LIN {X 0,Y 529.01,Z 397.613,A -85,B 0,C 180,E1 4371.131,E2 4371.131} C_VEL
LIN {X 0,Y 529.22,Z 392.744,A -85,B 0,C 180,E1 4373.977,E2 4373.977} C_VEL
LIN {X 0,Y 529.564,Z 381.839,A -85,B 0,C 180,E1 4376.861,E2 4376.861} C_VEL
LIN {X 0,Y 530.019,Z 365.768,A -85,B 0,C 180,E1 4379.389,E2 4379.389} C_VEL
LIN {X 0,Y 530.692,Z 344.7,A -85,B 0,C 180,E1 4381.518,E2 4381.518} C_VEL
LIN {X 0,Y 531.24,Z 320.224,A -85,B 0,C 180,E1 4383.087,E2 4383.087} C_VEL
LIN {X 0,Y 530.045,Z 304.294,A -85,B 0,C 180,E1 4383.791,E2 4383.791} C_VEL
LIN {X 0,Y 528.638,Z 297.81,A -85,B 0,C 180,E1 4384.104,E2 4384.104} C_VEL
LIN {X 0,Y 528.492,Z 297.81,A -85,B 0,C 180,E1 4390.468,E2 4390.468} C_VEL
LIN {X 0,Y 528.252,Z 297.81,A -85,B 0,C 180,E1 4395.103,E2 4395.103} C_VEL
LIN {X 0,Y 528.481,Z 297.81,A -85,B 0,C 180,E1 4400.136,E2 4400.136} C_VEL
LIN {X 0,Y 528.543,Z 297.81,A -85,B 0,C 180,E1 4402,E2 4402} C_VEL
LIN {X 0,Y 531.152,Z 316.99,A -85,B 0,C 180,E1 4402.758,E2 4402.758} C_VEL
LIN {X 0,Y 530.693,Z 340.931,A -85,B 0,C 180,E1 4404.146,E2 4404.146} C_VEL
LIN {X 0,Y 530.077,Z 362.098,A -85,B 0,C 180,E1 4406.102,E2 4406.102} C_VEL
LIN {X 0,Y 529.641,Z 379.29,A -85,B 0,C 180,E1 4408.572,E2 4408.572} C_VEL
LIN {X 0,Y 529.309,Z 390.67,A -85,B 0,C 180,E1 4411.226,E2 4411.226} C_VEL
LIN {X 0,Y 529.244,Z 396.059,A -85,B 0,C 180,E1 4413.495,E2 4413.495} C_VEL
LIN {X 0,Y 529.086,Z 397.913,A -85,B 0,C 180,E1 4416.551,E2 4416.551} C_VEL
LIN {X 0,Y 529.245,Z 394.993,A -85,B 0,C 180,E1 4419.023,E2 4419.023} C_VEL
LIN {X 0,Y 529.429,Z 386.158,A -85,B 0,C 180,E1 4421.926,E2 4421.926} C_VEL
LIN {X 0,Y 529.791,Z 372.114,A -85,B 0,C 180,E1 4424.519,E2 4424.519} C_VEL
LIN {X 0,Y 530.286,Z 353.941,A -85,B 0,C 180,E1 4426.675,E2 4426.675} C_VEL
LIN {X 0,Y 530.924,Z 331.466,A -85,B 0,C 180,E1 4428.405,E2 4428.405} C_VEL
LIN {X 0,Y 530.572,Z 307.156,A -85,B 0,C 180,E1 4429.557,E2 4429.557} C_VEL
LIN {X 0,Y 528.62,Z 297.81,A -85,B 0,C 180,E1 4429.894,E2 4429.894} C_VEL
LIN {X 0,Y 528.216,Z 297.81,A -85,B 0,C 180,E1 4435.374,E2 4435.374} C_VEL
LIN {X 0,Y 528.104,Z 297.81,A -85,B 0,C 180,E1 4440.972,E2 4440.972} C_VEL
LIN {X 0,Y 528.237,Z 297.81,A -85,B 0,C 180,E1 4446.863,E2 4446.863} C_VEL
LIN {X 0,Y 528.018,Z 297.81,A -85,B 0,C 180,E1 4451.992,E2 4451.992} C_VEL
LIN {X 0,Y 528.084,Z 297.81,A -85,B 0,C 180,E1 4457.984,E2 4457.984} C_VEL
LIN {X 0,Y 528.182,Z 297.81,A -85,B 0,C 180,E1 4463.126,E2 4463.126} C_VEL
LIN {X 0,Y 528.097,Z 297.81,A -85,B 0,C 180,E1 4469.034,E2 4469.034} C_VEL
LIN {X 0,Y 528.212,Z 297.81,A -85,B 0,C 180,E1 4474.614,E2 4474.614} C_VEL
LIN {X 0,Y 528.506,Z 297.81,A -85,B 0,C 180,E1 4480.429,E2 4480.429} C_VEL
LIN {X 0,Y 528.221,Z 297.81,A -85,B 0,C 180,E1 4486.241,E2 4486.241} C_VEL
LIN {X 0,Y 528.457,Z 297.81,A -85,B 0,C 180,E1 4491.781,E2 4491.781} C_VEL
LIN {X 0,Y 528.654,Z 297.81,A -85,B 0,C 180,E1 4497.505,E2 4497.505} C_VEL
LIN {X 0,Y 528.738,Z 297.81,A -85,B 0,C 180,E1 4503.262,E2 4503.262} C_VEL
LIN {X 0,Y 528.535,Z 297.81,A -85,B 0,C 180,E1 4509.854,E2 4509.854} C_VEL
LIN {X 0,Y 528.47,Z 297.81,A -85,B 0,C 180,E1 4514.881,E2 4514.881} C_VEL
LIN {X 0,Y 528.387,Z 297.81,A -85,B 0,C 180,E1 4520.031,E2 4520.031} C_VEL
LIN {X 0,Y 528.213,Z 297.81,A -85,B 0,C 180,E1 4525.363,E2 4525.363} C_VEL
LIN {X 0,Y 528.113,Z 297.81,A -85,B 0,C 180,E1 4530.531,E2 4530.531} C_VEL
LIN {X 0,Y 525.63,Z 297.81,A -85,B 0,C 180,E1 4531.933,E2 4531.933} C_VEL
LIN {X 0,Y 520.125,Z 297.81,A -85,B 0,C 180,E1 4534.278,E2 4534.278} C_VEL
LIN {X 0,Y 520.117,Z 297.81,A -85,B 0,C 180,E1 4539.652,E2 4539.652} C_VEL
LIN {X 0,Y 520.204,Z 297.81,A -85,B 0,C 180,E1 4545.878,E2 4545.878} C_VEL
LIN {X 0,Y 520.222,Z 297.81,A -85,B 0,C 180,E1 4551.539,E2 4551.539} C_VEL
LIN {X 0,Y 520.219,Z 297.81,A -85,B 0,C 180,E1 4557.251,E2 4557.251} C_VEL
LIN {X 0,Y 520.326,Z 297.81,A -85,B 0,C 180,E1 4562.353,E2 4562.353} C_VEL
LIN {X 0,Y 520.675,Z 298.125,A -85,B 0,C 180,E1 4565.62,E2 4565.62} C_VEL
LIN {X 0,Y 526.8,Z 321.24,A -85,B 0,C 180,E1 4566.185,E2 4566.185} C_VEL
LIN {X 0,Y 526.441,Z 376.223,A -85,B 0,C 180,E1 4567.058,E2 4567.058} C_VEL
LIN {X 0,Y 525.477,Z 410.152,A -85,B 0,C 180,E1 4568.241,E2 4568.241} C_VEL
LIN {X 0,Y 524.336,Z 441.478,A -85,B 0,C 180,E1 4570.016,E2 4570.016} C_VEL
LIN {X 0,Y 523.111,Z 470.478,A -85,B 0,C 180,E1 4572.38,E2 4572.38} C_VEL
LIN {X 0,Y 522.191,Z 495.428,A -85,B 0,C 180,E1 4575.203,E2 4575.203} C_VEL
LIN {X 0,Y 521.522,Z 516.3,A -85,B 0,C 180,E1 4578.51,E2 4578.51} C_VEL
LIN {X 0,Y 521.221,Z 531.706,A -85,B 0,C 180,E1 4582.095,E2 4582.095} C_VEL
LIN {X 0,Y 521.031,Z 539.685,A -85,B 0,C 180,E1 4585.015,E2 4585.015} C_VEL
LIN {X 0,Y 521.006,Z 544.24,A -85,B 0,C 180,E1 4588.34,E2 4588.34} C_VEL
LIN {X 0,Y 520.971,Z 544.236,A -85,B 0,C 180,E1 4591.659,E2 4591.659} C_VEL
LIN {X 0,Y 521.021,Z 539.682,A -85,B 0,C 180,E1 4594.984,E2 4594.984} C_VEL
LIN {X 0,Y 521.209,Z 530.265,A -85,B 0,C 180,E1 4598.323,E2 4598.323} C_VEL
LIN {X 0,Y 521.624,Z 514.044,A -85,B 0,C 180,E1 4601.894,E2 4601.894} C_VEL
LIN {X 0,Y 522.277,Z 493.101,A -85,B 0,C 180,E1 4605.072,E2 4605.072} C_VEL
LIN {X 0,Y 523.261,Z 467.062,A -85,B 0,C 180,E1 4607.915,E2 4607.915} C_VEL
LIN {X 0,Y 524.393,Z 437.782,A -85,B 0,C 180,E1 4610.2,E2 4610.2} C_VEL
LIN {X 0,Y 525.536,Z 405.635,A -85,B 0,C 180,E1 4611.917,E2 4611.917} C_VEL
LIN {X 0,Y 526.377,Z 372.12,A -85,B 0,C 180,E1 4613.008,E2 4613.008} C_VEL
LIN {X 0,Y 525.973,Z 316.706,A -85,B 0,C 180,E1 4613.869,E2 4613.869} C_VEL
LIN {X 0,Y 520.479,Z 297.81,A -85,B 0,C 180,E1 4614.412,E2 4614.412} C_VEL
LIN {X 0,Y 520.259,Z 297.81,A -85,B 0,C 180,E1 4619.543,E2 4619.543} C_VEL
LIN {X 0,Y 520.139,Z 297.81,A -85,B 0,C 180,E1 4625.466,E2 4625.466} C_VEL
LIN {X 0,Y 520.039,Z 297.81,A -85,B 0,C 180,E1 4631.865,E2 4631.865} C_VEL
LIN {X 0,Y 520.153,Z 297.81,A -85,B 0,C 180,E1 4638.158,E2 4638.158} C_VEL
LIN {X 0,Y 520.152,Z 297.81,A -85,B 0,C 180,E1 4644.32,E2 4644.32} C_VEL
LIN {X 0,Y 520.201,Z 297.81,A -85,B 0,C 180,E1 4650.485,E2 4650.485} C_VEL
LIN {X 0,Y 520.303,Z 297.81,A -85,B 0,C 180,E1 4656.055,E2 4656.055} C_VEL
LIN {X 0,Y 520.5,Z 297.81,A -85,B 0,C 180,E1 4661.414,E2 4661.414} C_VEL
LIN {X 0,Y 520.421,Z 297.81,A -85,B 0,C 180,E1 4668.3,E2 4668.3} C_VEL
LIN {X 0,Y 520.718,Z 297.81,A -85,B 0,C 180,E1 4673.354,E2 4673.354} C_VEL
LIN {X 0,Y 520.91,Z 297.81,A -85,B 0,C 180,E1 4678.35,E2 4678.35} C_VEL
LIN {X 0,Y 520.643,Z 297.81,A -85,B 0,C 180,E1 4684.999,E2 4684.999} C_VEL
LIN {X 0,Y 520.578,Z 297.81,A -85,B 0,C 180,E1 4690.027,E2 4690.027} C_VEL
LIN {X 0,Y 520.517,Z 297.81,A -85,B 0,C 180,E1 4695.135,E2 4695.135} C_VEL
LIN {X 0,Y 520.433,Z 297.81,A -85,B 0,C 180,E1 4700.373,E2 4700.373} C_VEL
LIN {X 0,Y 520.256,Z 297.81,A -85,B 0,C 180,E1 4705.955,E2 4705.955} C_VEL
LIN {X 0,Y 520.29,Z 297.81,A -85,B 0,C 180,E1 4711.483,E2 4711.483} C_VEL
LIN {X 0,Y 520.578,Z 298.037,A -85,B 0,C 180,E1 4715.507,E2 4715.507} C_VEL
LIN {X 0,Y 523.972,Z 316.712,A -85,B 0,C 180,E1 4716.32,E2 4716.32} C_VEL
LIN {X 0,Y 523.373,Z 340.806,A -85,B 0,C 180,E1 4717.743,E2 4717.743} C_VEL
LIN {X 0,Y 522.627,Z 362.011,A -85,B 0,C 180,E1 4719.712,E2 4719.712} C_VEL
LIN {X 0,Y 521.968,Z 378.391,A -85,B 0,C 180,E1 4722.011,E2 4722.011} C_VEL
LIN {X 0,Y 521.642,Z 390.294,A -85,B 0,C 180,E1 4724.63,E2 4724.63} C_VEL
LIN {X 0,Y 521.367,Z 396.709,A -85,B 0,C 180,E1 4727.1,E2 4727.1} C_VEL
LIN {X 0,Y 521.199,Z 398.827,A -85,B 0,C 180,E1 4728.848,E2 4728.848} C_VEL
LIN {X 0,Y 521.219,Z 398.452,A -85,B 0,C 180,E1 4731.434,E2 4731.434} C_VEL
LIN {X 0,Y 521.445,Z 393.523,A -85,B 0,C 180,E1 4734.144,E2 4734.144} C_VEL
LIN {X 0,Y 521.801,Z 382.63,A -85,B 0,C 180,E1 4737.02,E2 4737.02} C_VEL
LIN {X 0,Y 522.351,Z 366.237,A -85,B 0,C 180,E1 4739.61,E2 4739.61} C_VEL
LIN {X 0,Y 523.068,Z 345.175,A -85,B 0,C 180,E1 4741.748,E2 4741.748} C_VEL
LIN {X 0,Y 523.675,Z 320.982,A -85,B 0,C 180,E1 4743.315,E2 4743.315} C_VEL
LIN {X 0,Y 522.902,Z 307.36,A -85,B 0,C 180,E1 4743.938,E2 4743.938} C_VEL
LIN {X 0,Y 520.694,Z 297.81,A -85,B 0,C 180,E1 4744.349,E2 4744.349} C_VEL
LIN {X 0,Y 520.569,Z 297.81,A -85,B 0,C 180,E1 4751.406,E2 4751.406} C_VEL
LIN {X 0,Y 520.297,Z 297.81,A -85,B 0,C 180,E1 4756.584,E2 4756.584} C_VEL
LIN {X 0,Y 520.617,Z 297.81,A -85,B 0,C 180,E1 4761.772,E2 4761.772} C_VEL
LIN {X 0,Y 523.523,Z 317.705,A -85,B 0,C 180,E1 4762.548,E2 4762.548} C_VEL
LIN {X 0,Y 523.021,Z 342.35,A -85,B 0,C 180,E1 4763.997,E2 4763.997} C_VEL
LIN {X 0,Y 522.35,Z 363.931,A -85,B 0,C 180,E1 4766.044,E2 4766.044} C_VEL
LIN {X 0,Y 521.869,Z 380.844,A -85,B 0,C 180,E1 4768.551,E2 4768.551} C_VEL
LIN {X 0,Y 521.508,Z 392.014,A -85,B 0,C 180,E1 4771.244,E2 4771.244} C_VEL
LIN {X 0,Y 521.419,Z 396.902,A -85,B 0,C 180,E1 4773.319,E2 4773.319} C_VEL
LIN {X 0,Y 521.321,Z 398.774,A -85,B 0,C 180,E1 4774.982,E2 4774.982} C_VEL
LIN {X 0,Y 521.261,Z 398.955,A -85,B 0,C 180,E1 4776.65,E2 4776.65} C_VEL
LIN {X 0,Y 521.434,Z 395.894,A -85,B 0,C 180,E1 4779.159,E2 4779.159} C_VEL
LIN {X 0,Y 521.672,Z 386.873,A -85,B 0,C 180,E1 4782.106,E2 4782.106} C_VEL
LIN {X 0,Y 522.159,Z 371.912,A -85,B 0,C 180,E1 4784.836,E2 4784.836} C_VEL
LIN {X 0,Y 522.686,Z 353.038,A -85,B 0,C 180,E1 4787.024,E2 4787.024} C_VEL
LIN {X 0,Y 523.379,Z 330.241,A -85,B 0,C 180,E1 4788.723,E2 4788.723} C_VEL
LIN {X 0,Y 522.71,Z 307.361,A -85,B 0,C 180,E1 4789.796,E2 4789.796} C_VEL
LIN {X 0,Y 520.62,Z 297.81,A -85,B 0,C 180,E1 4790.235,E2 4790.235} C_VEL
LIN {X 0,Y 520.245,Z 297.81,A -85,B 0,C 180,E1 4795.923,E2 4795.923} C_VEL
LIN {X 0,Y 520.165,Z 297.81,A -85,B 0,C 180,E1 4801.479,E2 4801.479} C_VEL
LIN {X 0,Y 520.245,Z 297.81,A -85,B 0,C 180,E1 4807.526,E2 4807.526} C_VEL
LIN {X 0,Y 520.105,Z 297.81,A -85,B 0,C 180,E1 4813.486,E2 4813.486} C_VEL
LIN {X 0,Y 520.187,Z 297.81,A -85,B 0,C 180,E1 4818.959,E2 4818.959} C_VEL
LIN {X 0,Y 520.152,Z 297.81,A -85,B 0,C 180,E1 4824.52,E2 4824.52} C_VEL
LIN {X 0,Y 520.174,Z 297.81,A -85,B 0,C 180,E1 4830.493,E2 4830.493} C_VEL
LIN {X 0,Y 520.306,Z 297.81,A -85,B 0,C 180,E1 4836.032,E2 4836.032} C_VEL
LIN {X 0,Y 520.586,Z 297.81,A -85,B 0,C 180,E1 4841.395,E2 4841.395} C_VEL
LIN {X 0,Y 520.486,Z 297.81,A -85,B 0,C 180,E1 4848.28,E2 4848.28} C_VEL
LIN {X 0,Y 520.745,Z 297.81,A -85,B 0,C 180,E1 4853.333,E2 4853.333} C_VEL
LIN {X 0,Y 520.795,Z 297.81,A -85,B 0,C 180,E1 4859.99,E2 4859.99} C_VEL
LIN {X 0,Y 520.709,Z 297.81,A -85,B 0,C 180,E1 4864.977,E2 4864.977} C_VEL
LIN {X 0,Y 520.623,Z 297.81,A -85,B 0,C 180,E1 4870.005,E2 4870.005} C_VEL
LIN {X 0,Y 520.53,Z 297.81,A -85,B 0,C 180,E1 4875.114,E2 4875.114} C_VEL
LIN {X 0,Y 520.446,Z 297.81,A -85,B 0,C 180,E1 4880.35,E2 4880.35} C_VEL
LIN {X 0,Y 520.251,Z 297.81,A -85,B 0,C 180,E1 4885.951,E2 4885.951} C_VEL
LIN {X 0,Y 520.213,Z 297.81,A -85,B 0,C 180,E1 4891.464,E2 4891.464} C_VEL
LIN {X 0,Y 520.125,Z 297.81,A -85,B 0,C 180,E1 4894.278,E2 4894.278} C_VEL
LIN {X 0,Y 516.075,Z 297.81,A -85,B 0,C 180,E1 4896.161,E2 4896.161} C_VEL
LIN {X 0,Y 512.172,Z 297.81,A -85,B 0,C 180,E1 4898.073,E2 4898.073} C_VEL
LIN {X 0,Y 512.19,Z 297.81,A -85,B 0,C 180,E1 4902.645,E2 4902.645} C_VEL
LIN {X 0,Y 512.284,Z 297.81,A -85,B 0,C 180,E1 4907.413,E2 4907.413} C_VEL
LIN {X 0,Y 512.304,Z 297.81,A -85,B 0,C 180,E1 4912.667,E2 4912.667} C_VEL
LIN {X 0,Y 512.352,Z 297.81,A -85,B 0,C 180,E1 4918.645,E2 4918.645} C_VEL
LIN {X 0,Y 512.71,Z 298.24,A -85,B 0,C 180,E1 4925.299,E2 4925.299} C_VEL
LIN {X 0,Y 519.346,Z 322.362,A -85,B 0,C 180,E1 4925.909,E2 4925.909} C_VEL
LIN {X 0,Y 518.905,Z 377.073,A -85,B 0,C 180,E1 4926.808,E2 4926.808} C_VEL
LIN {X 0,Y 517.865,Z 410.624,A -85,B 0,C 180,E1 4928.019,E2 4928.019} C_VEL
LIN {X 0,Y 516.643,Z 441.524,A -85,B 0,C 180,E1 4929.817,E2 4929.817} C_VEL
LIN {X 0,Y 515.288,Z 470.21,A -85,B 0,C 180,E1 4932.211,E2 4932.211} C_VEL
LIN {X 0,Y 514.317,Z 495.586,A -85,B 0,C 180,E1 4935.164,E2 4935.164} C_VEL
LIN {X 0,Y 513.638,Z 516.351,A -85,B 0,C 180,E1 4938.562,E2 4938.562} C_VEL
LIN {X 0,Y 513.368,Z 530.59,A -85,B 0,C 180,E1 4941.974,E2 4941.974} C_VEL
LIN {X 0,Y 513.202,Z 538.59,A -85,B 0,C 180,E1 4944.939,E2 4944.939} C_VEL
LIN {X 0,Y 513.115,Z 543.397,A -85,B 0,C 180,E1 4948.693,E2 4948.693} C_VEL
LIN {X 0,Y 513.155,Z 543.151,A -85,B 0,C 180,E1 4951.685,E2 4951.685} C_VEL
LIN {X 0,Y 513.195,Z 538.562,A -85,B 0,C 180,E1 4955.06,E2 4955.06} C_VEL
LIN {X 0,Y 513.37,Z 529.098,A -85,B 0,C 180,E1 4958.451,E2 4958.451} C_VEL
LIN {X 0,Y 513.731,Z 512.805,A -85,B 0,C 180,E1 4962.08,E2 4962.08} C_VEL
LIN {X 0,Y 514.423,Z 491.759,A -85,B 0,C 180,E1 4965.307,E2 4965.307} C_VEL
LIN {X 0,Y 515.525,Z 465.567,A -85,B 0,C 180,E1 4968.193,E2 4968.193} C_VEL
LIN {X 0,Y 516.793,Z 436.098,A -85,B 0,C 180,E1 4970.511,E2 4970.511} C_VEL
LIN {X 0,Y 518.023,Z 403.441,A -85,B 0,C 180,E1 4972.252,E2 4972.252} C_VEL
LIN {X 0,Y 518.933,Z 370.14,A -85,B 0,C 180,E1 4973.318,E2 4973.318} C_VEL
LIN {X 0,Y 518.517,Z 318.414,A -85,B 0,C 180,E1 4974.129,E2 4974.129} C_VEL
LIN {X 0,Y 512.521,Z 297.81,A -85,B 0,C 180,E1 4974.719,E2 4974.719} C_VEL
LIN {X 0,Y 512.347,Z 297.81,A -85,B 0,C 180,E1 4981.354,E2 4981.354} C_VEL
LIN {X 0,Y 512.131,Z 297.81,A -85,B 0,C 180,E1 4987.307,E2 4987.307} C_VEL
LIN {X 0,Y 512.109,Z 297.81,A -85,B 0,C 180,E1 4992.665,E2 4992.665} C_VEL
LIN {X 0,Y 512.204,Z 297.81,A -85,B 0,C 180,E1 4997.435,E2 4997.435} C_VEL
LIN {X 0,Y 512.256,Z 297.81,A -85,B 0,C 180,E1 5002.689,E2 5002.689} C_VEL
LIN {X 0,Y 512.254,Z 297.81,A -85,B 0,C 180,E1 5008.679,E2 5008.679} C_VEL
LIN {X 0,Y 512.339,Z 297.81,A -85,B 0,C 180,E1 5013.792,E2 5013.792} C_VEL
LIN {X 0,Y 512.511,Z 297.81,A -85,B 0,C 180,E1 5019.32,E2 5019.32} C_VEL
LIN {X 0,Y 512.4,Z 297.81,A -85,B 0,C 180,E1 5024.641,E2 5024.641} C_VEL
LIN {X 0,Y 512.583,Z 297.81,A -85,B 0,C 180,E1 5029.837,E2 5029.837} C_VEL
LIN {X 0,Y 512.823,Z 297.81,A -85,B 0,C 180,E1 5034.946,E2 5034.946} C_VEL
LIN {X 0,Y 512.843,Z 297.81,A -85,B 0,C 180,E1 5040.011,E2 5040.011} C_VEL
LIN {X 0,Y 512.762,Z 297.81,A -85,B 0,C 180,E1 5045.076,E2 5045.076} C_VEL
LIN {X 0,Y 512.654,Z 297.81,A -85,B 0,C 180,E1 5050.183,E2 5050.183} C_VEL
LIN {X 0,Y 512.587,Z 297.81,A -85,B 0,C 180,E1 5055.375,E2 5055.375} C_VEL
LIN {X 0,Y 512.506,Z 297.81,A -85,B 0,C 180,E1 5060.703,E2 5060.703} C_VEL
LIN {X 0,Y 512.341,Z 297.81,A -85,B 0,C 180,E1 5066.231,E2 5066.231} C_VEL
LIN {X 0,Y 512.41,Z 297.81,A -85,B 0,C 180,E1 5072.025,E2 5072.025} C_VEL
LIN {X 0,Y 512.641,Z 298.471,A -85,B 0,C 180,E1 5075.21,E2 5075.21} C_VEL
LIN {X 0,Y 516.466,Z 317.44,A -85,B 0,C 180,E1 5076.066,E2 5076.066} C_VEL
LIN {X 0,Y 515.779,Z 342.453,A -85,B 0,C 180,E1 5077.579,E2 5077.579} C_VEL
LIN {X 0,Y 514.948,Z 364.18,A -85,B 0,C 180,E1 5079.664,E2 5079.664} C_VEL
LIN {X 0,Y 514.207,Z 381.651,A -85,B 0,C 180,E1 5082.269,E2 5082.269} C_VEL
LIN {X 0,Y 513.815,Z 393.456,A -85,B 0,C 180,E1 5085.184,E2 5085.184} C_VEL
LIN {X 0,Y 513.528,Z 398.509,A -85,B 0,C 180,E1 5087.48,E2 5087.48} C_VEL
LIN {X 0,Y 513.351,Z 400.277,A -85,B 0,C 180,E1 5089.861,E2 5089.861} C_VEL
LIN {X 0,Y 513.497,Z 398.191,A -85,B 0,C 180,E1 5092.528,E2 5092.528} C_VEL
LIN {X 0,Y 513.823,Z 391.142,A -85,B 0,C 180,E1 5095.337,E2 5095.337} C_VEL
LIN {X 0,Y 514.248,Z 378.399,A -85,B 0,C 180,E1 5098.118,E2 5098.118} C_VEL
LIN {X 0,Y 514.879,Z 361.217,A -85,B 0,C 180,E1 5100.486,E2 5100.486} C_VEL
LIN {X 0,Y 515.658,Z 339.32,A -85,B 0,C 180,E1 5102.475,E2 5102.475} C_VEL
LIN {X 0,Y 516.265,Z 313.576,A -85,B 0,C 180,E1 5103.932,E2 5103.932} C_VEL
LIN {X 0,Y 512.751,Z 297.81,A -85,B 0,C 180,E1 5104.624,E2 5104.624} C_VEL
LIN {X 0,Y 512.621,Z 297.81,A -85,B 0,C 180,E1 5111.107,E2 5111.107} C_VEL
LIN {X 0,Y 512.4,Z 297.81,A -85,B 0,C 180,E1 5116.422,E2 5116.422} C_VEL
LIN {X 0,Y 512.681,Z 298.165,A -85,B 0,C 180,E1 5121.538,E2 5121.538} C_VEL
LIN {X 0,Y 515.915,Z 317.156,A -85,B 0,C 180,E1 5122.279,E2 5122.279} C_VEL
LIN {X 0,Y 515.399,Z 341.774,A -85,B 0,C 180,E1 5123.697,E2 5123.697} C_VEL
LIN {X 0,Y 514.723,Z 363.188,A -85,B 0,C 180,E1 5125.685,E2 5125.685} C_VEL
LIN {X 0,Y 514.138,Z 380.136,A -85,B 0,C 180,E1 5128.108,E2 5128.108} C_VEL
LIN {X 0,Y 513.759,Z 392.065,A -85,B 0,C 180,E1 5130.842,E2 5130.842} C_VEL
LIN {X 0,Y 513.602,Z 398.133,A -85,B 0,C 180,E1 5133.369,E2 5133.369} C_VEL
LIN {X 0,Y 513.489,Z 399.907,A -85,B 0,C 180,E1 5135.058,E2 5135.058} C_VEL
LIN {X 0,Y 513.453,Z 399.98,A -85,B 0,C 180,E1 5136.752,E2 5136.752} C_VEL
LIN {X 0,Y 513.644,Z 396.777,A -85,B 0,C 180,E1 5139.299,E2 5139.299} C_VEL
LIN {X 0,Y 513.902,Z 387.561,A -85,B 0,C 180,E1 5142.292,E2 5142.292} C_VEL
LIN {X 0,Y 514.46,Z 372.567,A -85,B 0,C 180,E1 5145.03,E2 5145.03} C_VEL
LIN {X 0,Y 515.043,Z 353.66,A -85,B 0,C 180,E1 5147.234,E2 5147.234} C_VEL
LIN {X 0,Y 515.789,Z 329.997,A -85,B 0,C 180,E1 5148.993,E2 5148.993} C_VEL
LIN {X 0,Y 515.319,Z 309.758,A -85,B 0,C 180,E1 5149.949,E2 5149.949} C_VEL
LIN {X 0,Y 512.662,Z 297.81,A -85,B 0,C 180,E1 5150.458,E2 5150.458} C_VEL
LIN {X 0,Y 512.318,Z 297.81,A -85,B 0,C 180,E1 5156.22,E2 5156.22} C_VEL
LIN {X 0,Y 512.242,Z 297.81,A -85,B 0,C 180,E1 5162.023,E2 5162.023} C_VEL
LIN {X 0,Y 512.345,Z 297.81,A -85,B 0,C 180,E1 5168.208,E2 5168.208} C_VEL
LIN {X 0,Y 512.173,Z 297.81,A -85,B 0,C 180,E1 5175,E2 5175} C_VEL
LIN {X 0,Y 512.313,Z 297.81,A -85,B 0,C 180,E1 5179.981,E2 5179.981} C_VEL
LIN {X 0,Y 512.19,Z 297.81,A -85,B 0,C 180,E1 5185.946,E2 5185.946} C_VEL
LIN {X 0,Y 512.299,Z 297.81,A -85,B 0,C 180,E1 5192.088,E2 5192.088} C_VEL
LIN {X 0,Y 512.437,Z 297.81,A -85,B 0,C 180,E1 5197.48,E2 5197.48} C_VEL
LIN {X 0,Y 512.64,Z 297.81,A -85,B 0,C 180,E1 5202.869,E2 5202.869} C_VEL
LIN {X 0,Y 512.644,Z 297.81,A -85,B 0,C 180,E1 5209.816,E2 5209.816} C_VEL
LIN {X 0,Y 512.806,Z 297.81,A -85,B 0,C 180,E1 5214.925,E2 5214.925} C_VEL
LIN {X 0,Y 512.905,Z 297.81,A -85,B 0,C 180,E1 5219.989,E2 5219.989} C_VEL
LIN {X 0,Y 512.816,Z 297.81,A -85,B 0,C 180,E1 5225.054,E2 5225.054} C_VEL
LIN {X 0,Y 512.697,Z 297.81,A -85,B 0,C 180,E1 5230.161,E2 5230.161} C_VEL
LIN {X 0,Y 512.592,Z 297.81,A -85,B 0,C 180,E1 5235.353,E2 5235.353} C_VEL
LIN {X 0,Y 512.54,Z 297.81,A -85,B 0,C 180,E1 5240.679,E2 5240.679} C_VEL
LIN {X 0,Y 512.335,Z 297.81,A -85,B 0,C 180,E1 5246.208,E2 5246.208} C_VEL
LIN {X 0,Y 512.318,Z 297.81,A -85,B 0,C 180,E1 5252.006,E2 5252.006} C_VEL
LIN {X 0,Y 512.172,Z 297.81,A -85,B 0,C 180,E1 5258.073,E2 5258.073} C_VEL
LIN {X 0,Y 509.707,Z 297.81,A -85,B 0,C 180,E1 5259.503,E2 5259.503} C_VEL
LIN {X 0,Y 504.16,Z 297.81,A -85,B 0,C 180,E1 5261.894,E2 5261.894} C_VEL
LIN {X 0,Y 504.317,Z 297.81,A -85,B 0,C 180,E1 5268.407,E2 5268.407} C_VEL
LIN {X 0,Y 504.409,Z 297.81,A -85,B 0,C 180,E1 5273.86,E2 5273.86} C_VEL
LIN {X 0,Y 504.438,Z 297.81,A -85,B 0,C 180,E1 5280.153,E2 5280.153} C_VEL
LIN {X 0,Y 504.747,Z 297.81,A -85,B 0,C 180,E1 5284.956,E2 5284.956} C_VEL
LIN {X 0,Y 511.924,Z 323.416,A -85,B 0,C 180,E1 5285.626,E2 5285.626} C_VEL
LIN {X 0,Y 511.479,Z 375.275,A -85,B 0,C 180,E1 5286.481,E2 5286.481} C_VEL
LIN {X 0,Y 510.366,Z 408.077,A -85,B 0,C 180,E1 5287.649,E2 5287.649} C_VEL
LIN {X 0,Y 509.01,Z 439.986,A -85,B 0,C 180,E1 5289.501,E2 5289.501} C_VEL
LIN {X 0,Y 507.6,Z 468.31,A -85,B 0,C 180,E1 5291.873,E2 5291.873} C_VEL
LIN {X 0,Y 506.488,Z 493.927,A -85,B 0,C 180,E1 5294.866,E2 5294.866} C_VEL
LIN {X 0,Y 505.822,Z 514.054,A -85,B 0,C 180,E1 5298.164,E2 5298.164} C_VEL
LIN {X 0,Y 505.483,Z 529.47,A -85,B 0,C 180,E1 5301.848,E2 5301.848} C_VEL
LIN {X 0,Y 505.381,Z 537.5,A -85,B 0,C 180,E1 5304.86,E2 5304.86} C_VEL
LIN {X 0,Y 505.354,Z 542.074,A -85,B 0,C 180,E1 5308.288,E2 5308.288} C_VEL
LIN {X 0,Y 505.331,Z 542.053,A -85,B 0,C 180,E1 5311.711,E2 5311.711} C_VEL
LIN {X 0,Y 505.376,Z 537.442,A -85,B 0,C 180,E1 5315.139,E2 5315.139} C_VEL
LIN {X 0,Y 505.493,Z 527.923,A -85,B 0,C 180,E1 5318.584,E2 5318.584} C_VEL
LIN {X 0,Y 505.868,Z 511.57,A -85,B 0,C 180,E1 5322.271,E2 5322.271} C_VEL
LIN {X 0,Y 506.589,Z 490.419,A -85,B 0,C 180,E1 5325.55,E2 5325.55} C_VEL
LIN {X 0,Y 507.744,Z 465.056,A -85,B 0,C 180,E1 5328.389,E2 5328.389} C_VEL
LIN {X 0,Y 509.093,Z 435.995,A -85,B 0,C 180,E1 5330.722,E2 5330.722} C_VEL
LIN {X 0,Y 510.343,Z 404.919,A -85,B 0,C 180,E1 5332.437,E2 5332.437} C_VEL
LIN {X 0,Y 511.415,Z 371.198,A -85,B 0,C 180,E1 5333.573,E2 5333.573} C_VEL
LIN {X 0,Y 511.184,Z 320.255,A -85,B 0,C 180,E1 5334.39,E2 5334.39} C_VEL
LIN {X 0,Y 504.59,Z 297.81,A -85,B 0,C 180,E1 5334.987,E2 5334.987} C_VEL
LIN {X 0,Y 504.386,Z 297.81,A -85,B 0,C 180,E1 5340.57,E2 5340.57} C_VEL
LIN {X 0,Y 504.223,Z 297.81,A -85,B 0,C 180,E1 5346.765,E2 5346.765} C_VEL
LIN {X 0,Y 504.129,Z 297.81,A -85,B 0,C 180,E1 5353.507,E2 5353.507} C_VEL
LIN {X 0,Y 504.258,Z 297.81,A -85,B 0,C 180,E1 5358.838,E2 5358.838} C_VEL
LIN {X 0,Y 504.273,Z 297.81,A -85,B 0,C 180,E1 5365.362,E2 5365.362} C_VEL
LIN {X 0,Y 504.341,Z 297.81,A -85,B 0,C 180,E1 5371.409,E2 5371.409} C_VEL
LIN {X 0,Y 504.466,Z 297.81,A -85,B 0,C 180,E1 5377.127,E2 5377.127} C_VEL
LIN {X 0,Y 504.656,Z 297.81,A -85,B 0,C 180,E1 5383.105,E2 5383.105} C_VEL
LIN {X 0,Y 504.663,Z 297.81,A -85,B 0,C 180,E1 5389.675,E2 5389.675} C_VEL
LIN {X 0,Y 504.911,Z 297.81,A -85,B 0,C 180,E1 5394.867,E2 5394.867} C_VEL
LIN {X 0,Y 504.942,Z 297.81,A -85,B 0,C 180,E1 5400.011,E2 5400.011} C_VEL
LIN {X 0,Y 504.849,Z 297.81,A -85,B 0,C 180,E1 5405.156,E2 5405.156} C_VEL
LIN {X 0,Y 504.733,Z 297.81,A -85,B 0,C 180,E1 5410.345,E2 5410.345} C_VEL
LIN {X 0,Y 504.658,Z 297.81,A -85,B 0,C 180,E1 5415.623,E2 5415.623} C_VEL
LIN {X 0,Y 504.555,Z 297.81,A -85,B 0,C 180,E1 5421.044,E2 5421.044} C_VEL
LIN {X 0,Y 504.402,Z 297.81,A -85,B 0,C 180,E1 5426.676,E2 5426.676} C_VEL
LIN {X 0,Y 504.479,Z 297.81,A -85,B 0,C 180,E1 5433.12,E2 5433.12} C_VEL
LIN {X 0,Y 504.695,Z 297.81,A -85,B 0,C 180,E1 5434.859,E2 5434.859} C_VEL
LIN {X 0,Y 508.978,Z 319.273,A -85,B 0,C 180,E1 5435.856,E2 5435.856} C_VEL
LIN {X 0,Y 508.145,Z 344.738,A -85,B 0,C 180,E1 5437.458,E2 5437.458} C_VEL
LIN {X 0,Y 507.289,Z 364.971,A -85,B 0,C 180,E1 5439.448,E2 5439.448} C_VEL
LIN {X 0,Y 506.503,Z 381.252,A -85,B 0,C 180,E1 5441.858,E2 5441.858} C_VEL
LIN {X 0,Y 506.066,Z 393.334,A -85,B 0,C 180,E1 5444.691,E2 5444.691} C_VEL
LIN {X 0,Y 505.701,Z 399.732,A -85,B 0,C 180,E1 5447.524,E2 5447.524} C_VEL
LIN {X 0,Y 505.557,Z 401.108,A -85,B 0,C 180,E1 5448.955,E2 5448.955} C_VEL
LIN {X 0,Y 505.627,Z 400.168,A -85,B 0,C 180,E1 5451.92,E2 5451.92} C_VEL
LIN {X 0,Y 505.998,Z 393.249,A -85,B 0,C 180,E1 5455.105,E2 5455.105} C_VEL
LIN {X 0,Y 506.455,Z 381.46,A -85,B 0,C 180,E1 5457.885,E2 5457.885} C_VEL
LIN {X 0,Y 507.129,Z 364.702,A -85,B 0,C 180,E1 5460.371,E2 5460.371} C_VEL
LIN {X 0,Y 507.921,Z 343.239,A -85,B 0,C 180,E1 5462.46,E2 5462.46} C_VEL
LIN {X 0,Y 508.683,Z 318.395,A -85,B 0,C 180,E1 5463.993,E2 5463.993} C_VEL
LIN {X 0,Y 504.769,Z 297.81,A -85,B 0,C 180,E1 5464.964,E2 5464.964} C_VEL
LIN {X 0,Y 504.692,Z 297.81,A -85,B 0,C 180,E1 5470.799,E2 5470.799} C_VEL
LIN {X 0,Y 504.487,Z 297.81,A -85,B 0,C 180,E1 5476.156,E2 5476.156} C_VEL
LIN {X 0,Y 504.788,Z 297.81,A -85,B 0,C 180,E1 5481.269,E2 5481.269} C_VEL
LIN {X 0,Y 508.304,Z 319.015,A -85,B 0,C 180,E1 5482.109,E2 5482.109} C_VEL
LIN {X 0,Y 507.757,Z 344.013,A -85,B 0,C 180,E1 5483.602,E2 5483.602} C_VEL
LIN {X 0,Y 506.99,Z 365.242,A -85,B 0,C 180,E1 5485.646,E2 5485.646} C_VEL
LIN {X 0,Y 506.375,Z 381.686,A -85,B 0,C 180,E1 5488.079,E2 5488.079} C_VEL
LIN {X 0,Y 505.975,Z 393.428,A -85,B 0,C 180,E1 5490.855,E2 5490.855} C_VEL
LIN {X 0,Y 505.772,Z 399.345,A -85,B 0,C 180,E1 5493.421,E2 5493.421} C_VEL
LIN {X 0,Y 505.659,Z 401.04,A -85,B 0,C 180,E1 5495.137,E2 5495.137} C_VEL
LIN {X 0,Y 505.628,Z 401.008,A -85,B 0,C 180,E1 5496.857,E2 5496.857} C_VEL
LIN {X 0,Y 505.848,Z 397.885,A -85,B 0,C 180,E1 5499.338,E2 5499.338} C_VEL
LIN {X 0,Y 506.095,Z 389.997,A -85,B 0,C 180,E1 5502.048,E2 5502.048} C_VEL
LIN {X 0,Y 506.562,Z 377.081,A -85,B 0,C 180,E1 5504.645,E2 5504.645} C_VEL
LIN {X 0,Y 507.24,Z 358.022,A -85,B 0,C 180,E1 5507.084,E2 5507.084} C_VEL
LIN {X 0,Y 508.037,Z 335.925,A -85,B 0,C 180,E1 5508.897,E2 5508.897} C_VEL
LIN {X 0,Y 507.724,Z 311.142,A -85,B 0,C 180,E1 5510.154,E2 5510.154} C_VEL
LIN {X 0,Y 504.732,Z 297.81,A -85,B 0,C 180,E1 5510.771,E2 5510.771} C_VEL
LIN {X 0,Y 504.378,Z 297.81,A -85,B 0,C 180,E1 5516.665,E2 5516.665} C_VEL
LIN {X 0,Y 504.268,Z 297.81,A -85,B 0,C 180,E1 5523.06,E2 5523.06} C_VEL
LIN {X 0,Y 504.377,Z 297.81,A -85,B 0,C 180,E1 5528.924,E2 5528.924} C_VEL
LIN {X 0,Y 504.198,Z 297.81,A -85,B 0,C 180,E1 5535.914,E2 5535.914} C_VEL
LIN {X 0,Y 504.365,Z 297.81,A -85,B 0,C 180,E1 5541.068,E2 5541.068} C_VEL
LIN {X 0,Y 504.262,Z 297.81,A -85,B 0,C 180,E1 5547.395,E2 5547.395} C_VEL
LIN {X 0,Y 504.434,Z 297.81,A -85,B 0,C 180,E1 5553.825,E2 5553.825} C_VEL
LIN {X 0,Y 504.612,Z 297.81,A -85,B 0,C 180,E1 5558.958,E2 5558.958} C_VEL
LIN {X 0,Y 504.574,Z 297.81,A -85,B 0,C 180,E1 5564.374,E2 5564.374} C_VEL
LIN {X 0,Y 504.701,Z 297.81,A -85,B 0,C 180,E1 5570.634,E2 5570.634} C_VEL
LIN {X 0,Y 504.864,Z 297.81,A -85,B 0,C 180,E1 5576.562,E2 5576.562} C_VEL
LIN {X 0,Y 504.879,Z 297.81,A -85,B 0,C 180,E1 5581.702,E2 5581.702} C_VEL
LIN {X 0,Y 504.793,Z 297.81,A -85,B 0,C 180,E1 5586.857,E2 5586.857} C_VEL
LIN {X 0,Y 504.722,Z 297.81,A -85,B 0,C 180,E1 5592.07,E2 5592.07} C_VEL
LIN {X 0,Y 504.653,Z 297.81,A -85,B 0,C 180,E1 5597.388,E2 5597.388} C_VEL
LIN {X 0,Y 504.538,Z 297.81,A -85,B 0,C 180,E1 5602.87,E2 5602.87} C_VEL
LIN {X 0,Y 504.37,Z 297.81,A -85,B 0,C 180,E1 5608.589,E2 5608.589} C_VEL
LIN {X 0,Y 504.313,Z 297.81,A -85,B 0,C 180,E1 5614.635,E2 5614.635} C_VEL
LIN {X 0,Y 504.206,Z 297.81,A -85,B 0,C 180,E1 5621.167,E2 5621.167} C_VEL
LIN {X 0,Y 504.16,Z 297.81,A -85,B 0,C 180,E1 5621.894,E2 5621.894} C_VEL
LIN {X 0,Y 500.238,Z 297.81,A -85,B 0,C 180,E1 5623.843,E2 5623.843} C_VEL
LIN {X 0,Y 496.334,Z 297.81,A -85,B 0,C 180,E1 5625.822,E2 5625.822} C_VEL
LIN {X 0,Y 496.418,Z 297.81,A -85,B 0,C 180,E1 5632.202,E2 5632.202} C_VEL
LIN {X 0,Y 496.393,Z 297.81,A -85,B 0,C 180,E1 5638.322,E2 5638.322} C_VEL
LIN {X 0,Y 496.803,Z 298.216,A -85,B 0,C 180,E1 5644.628,E2 5644.628} C_VEL
LIN {X 0,Y 504.508,Z 324.918,A -85,B 0,C 180,E1 5645.344,E2 5645.344} C_VEL
LIN {X 0,Y 503.994,Z 375.595,A -85,B 0,C 180,E1 5646.203,E2 5646.203} C_VEL
LIN {X 0,Y 502.761,Z 409.193,A -85,B 0,C 180,E1 5647.442,E2 5647.442} C_VEL
LIN {X 0,Y 501.327,Z 440.03,A -85,B 0,C 180,E1 5649.287,E2 5649.287} C_VEL
LIN {X 0,Y 499.79,Z 468.763,A -85,B 0,C 180,E1 5651.767,E2 5651.767} C_VEL
LIN {X 0,Y 498.616,Z 493.769,A -85,B 0,C 180,E1 5654.778,E2 5654.778} C_VEL
LIN {X 0,Y 497.927,Z 514.022,A -85,B 0,C 180,E1 5658.196,E2 5658.196} C_VEL
LIN {X 0,Y 497.6,Z 528.354,A -85,B 0,C 180,E1 5661.717,E2 5661.717} C_VEL
LIN {X 0,Y 497.526,Z 536.405,A -85,B 0,C 180,E1 5664.779,E2 5664.779} C_VEL
LIN {X 0,Y 497.544,Z 540.988,A -85,B 0,C 180,E1 5668.262,E2 5668.262} C_VEL
LIN {X 0,Y 497.503,Z 540.955,A -85,B 0,C 180,E1 5671.738,E2 5671.738} C_VEL
LIN {X 0,Y 497.527,Z 536.317,A -85,B 0,C 180,E1 5675.22,E2 5675.22} C_VEL
LIN {X 0,Y 497.625,Z 525.604,A -85,B 0,C 180,E1 5679.031,E2 5679.031} C_VEL
LIN {X 0,Y 497.984,Z 509.141,A -85,B 0,C 180,E1 5682.69,E2 5682.69} C_VEL
LIN {X 0,Y 498.878,Z 487.416,A -85,B 0,C 180,E1 5686.022,E2 5686.022} C_VEL
LIN {X 0,Y 500.102,Z 460.646,A -85,B 0,C 180,E1 5688.958,E2 5688.958} C_VEL
LIN {X 0,Y 501.61,Z 431.169,A -85,B 0,C 180,E1 5691.254,E2 5691.254} C_VEL
LIN {X 0,Y 503.081,Z 399.031,A -85,B 0,C 180,E1 5692.95,E2 5692.95} C_VEL
LIN {X 0,Y 504.064,Z 365.317,A -85,B 0,C 180,E1 5693.986,E2 5693.986} C_VEL
LIN {X 0,Y 503.772,Z 321.929,A -85,B 0,C 180,E1 5694.666,E2 5694.666} C_VEL
LIN {X 0,Y 496.654,Z 297.81,A -85,B 0,C 180,E1 5695.357,E2 5695.357} C_VEL
LIN {X 0,Y 496.392,Z 297.81,A -85,B 0,C 180,E1 5701.677,E2 5701.677} C_VEL
LIN {X 0,Y 496.22,Z 297.81,A -85,B 0,C 180,E1 5707.768,E2 5707.768} C_VEL
LIN {X 0,Y 496.262,Z 297.81,A -85,B 0,C 180,E1 5714.375,E2 5714.375} C_VEL
LIN {X 0,Y 496.345,Z 297.81,A -85,B 0,C 180,E1 5720.337,E2 5720.337} C_VEL
LIN {X 0,Y 496.331,Z 297.81,A -85,B 0,C 180,E1 5726.833,E2 5726.833} C_VEL
LIN {X 0,Y 496.443,Z 297.81,A -85,B 0,C 180,E1 5732.886,E2 5732.886} C_VEL
LIN {X 0,Y 496.624,Z 297.81,A -85,B 0,C 180,E1 5738.627,E2 5738.627} C_VEL
LIN {X 0,Y 496.62,Z 297.81,A -85,B 0,C 180,E1 5744.14,E2 5744.14} C_VEL
LIN {X 0,Y 496.732,Z 297.81,A -85,B 0,C 180,E1 5749.509,E2 5749.509} C_VEL
LIN {X 0,Y 497.012,Z 297.81,A -85,B 0,C 180,E1 5754.785,E2 5754.785} C_VEL
LIN {X 0,Y 497.05,Z 297.81,A -85,B 0,C 180,E1 5760.011,E2 5760.011} C_VEL
LIN {X 0,Y 496.955,Z 297.81,A -85,B 0,C 180,E1 5765.238,E2 5765.238} C_VEL
LIN {X 0,Y 496.81,Z 297.81,A -85,B 0,C 180,E1 5770.512,E2 5770.512} C_VEL
LIN {X 0,Y 496.745,Z 297.81,A -85,B 0,C 180,E1 5775.878,E2 5775.878} C_VEL
LIN {X 0,Y 496.636,Z 297.81,A -85,B 0,C 180,E1 5781.396,E2 5781.396} C_VEL
LIN {X 0,Y 496.445,Z 297.81,A -85,B 0,C 180,E1 5787.139,E2 5787.139} C_VEL
LIN {X 0,Y 496.605,Z 297.81,A -85,B 0,C 180,E1 5793.715,E2 5793.715} C_VEL
LIN {X 0,Y 496.787,Z 298.558,A -85,B 0,C 180,E1 5794.556,E2 5794.556} C_VEL
LIN {X 0,Y 501.482,Z 320.249,A -85,B 0,C 180,E1 5795.595,E2 5795.595} C_VEL
LIN {X 0,Y 500.606,Z 345.075,A -85,B 0,C 180,E1 5797.176,E2 5797.176} C_VEL
LIN {X 0,Y 499.649,Z 365.838,A -85,B 0,C 180,E1 5799.235,E2 5799.235} C_VEL
LIN {X 0,Y 498.774,Z 382.507,A -85,B 0,C 180,E1 5801.744,E2 5801.744} C_VEL
LIN {X 0,Y 498.319,Z 394.182,A -85,B 0,C 180,E1 5804.514,E2 5804.514} C_VEL
LIN {X 0,Y 497.889,Z 400.829,A -85,B 0,C 180,E1 5807.472,E2 5807.472} C_VEL
LIN {X 0,Y 497.717,Z 402.362,A -85,B 0,C 180,E1 5810.456,E2 5810.456} C_VEL
LIN {X 0,Y 497.924,Z 399.5,A -85,B 0,C 180,E1 5813.101,E2 5813.101} C_VEL
LIN {X 0,Y 498.304,Z 391.515,A -85,B 0,C 180,E1 5816.011,E2 5816.011} C_VEL
LIN {X 0,Y 498.845,Z 378.164,A -85,B 0,C 180,E1 5818.778,E2 5818.778} C_VEL
LIN {X 0,Y 499.727,Z 359.301,A -85,B 0,C 180,E1 5821.277,E2 5821.277} C_VEL
LIN {X 0,Y 500.651,Z 336.506,A -85,B 0,C 180,E1 5823.242,E2 5823.242} C_VEL
LIN {X 0,Y 500.481,Z 312.872,A -85,B 0,C 180,E1 5824.555,E2 5824.555} C_VEL
LIN {X 0,Y 496.813,Z 297.81,A -85,B 0,C 180,E1 5825.324,E2 5825.324} C_VEL
LIN {X 0,Y 496.8,Z 297.81,A -85,B 0,C 180,E1 5832.318,E2 5832.318} C_VEL
LIN {X 0,Y 496.775,Z 297.81,A -85,B 0,C 180,E1 5839.499,E2 5839.499} C_VEL
LIN {X 0,Y 496.885,Z 297.81,A -85,B 0,C 180,E1 5841.025,E2 5841.025} C_VEL
LIN {X 0,Y 500.71,Z 320.718,A -85,B 0,C 180,E1 5841.934,E2 5841.934} C_VEL
LIN {X 0,Y 500.123,Z 344.755,A -85,B 0,C 180,E1 5843.395,E2 5843.395} C_VEL
LIN {X 0,Y 499.321,Z 365.955,A -85,B 0,C 180,E1 5845.451,E2 5845.451} C_VEL
LIN {X 0,Y 498.627,Z 383.213,A -85,B 0,C 180,E1 5848.049,E2 5848.049} C_VEL
LIN {X 0,Y 498.207,Z 393.69,A -85,B 0,C 180,E1 5850.532,E2 5850.532} C_VEL
LIN {X 0,Y 497.954,Z 400.541,A -85,B 0,C 180,E1 5853.475,E2 5853.475} C_VEL
LIN {X 0,Y 497.858,Z 402.168,A -85,B 0,C 180,E1 5855.218,E2 5855.218} C_VEL
LIN {X 0,Y 497.817,Z 402.036,A -85,B 0,C 180,E1 5856.965,E2 5856.965} C_VEL
LIN {X 0,Y 498.101,Z 397.679,A -85,B 0,C 180,E1 5859.992,E2 5859.992} C_VEL
LIN {X 0,Y 498.399,Z 388.938,A -85,B 0,C 180,E1 5862.681,E2 5862.681} C_VEL
LIN {X 0,Y 499.066,Z 374.187,A -85,B 0,C 180,E1 5865.398,E2 5865.398} C_VEL
LIN {X 0,Y 499.76,Z 354.95,A -85,B 0,C 180,E1 5867.678,E2 5867.678} C_VEL
LIN {X 0,Y 500.597,Z 331.578,A -85,B 0,C 180,E1 5869.443,E2 5869.443} C_VEL
LIN {X 0,Y 499.982,Z 311.767,A -85,B 0,C 180,E1 5870.407,E2 5870.407} C_VEL
LIN {X 0,Y 496.801,Z 297.81,A -85,B 0,C 180,E1 5870.93,E2 5870.93} C_VEL
LIN {X 0,Y 496.405,Z 297.81,A -85,B 0,C 180,E1 5877.128,E2 5877.128} C_VEL
LIN {X 0,Y 496.362,Z 297.81,A -85,B 0,C 180,E1 5883.177,E2 5883.177} C_VEL
LIN {X 0,Y 496.344,Z 297.81,A -85,B 0,C 180,E1 5889.677,E2 5889.677} C_VEL
LIN {X 0,Y 496.286,Z 297.81,A -85,B 0,C 180,E1 5895.609,E2 5895.609} C_VEL
LIN {X 0,Y 496.353,Z 297.81,A -85,B 0,C 180,E1 5900.309,E2 5900.309} C_VEL
LIN {X 0,Y 496.344,Z 297.81,A -85,B 0,C 180,E1 5906.808,E2 5906.808} C_VEL
LIN {X 0,Y 496.411,Z 297.81,A -85,B 0,C 180,E1 5912.859,E2 5912.859} C_VEL
LIN {X 0,Y 496.676,Z 297.81,A -85,B 0,C 180,E1 5918.606,E2 5918.606} C_VEL
LIN {X 0,Y 496.692,Z 297.81,A -85,B 0,C 180,E1 5924.12,E2 5924.12} C_VEL
LIN {X 0,Y 496.791,Z 297.81,A -85,B 0,C 180,E1 5929.488,E2 5929.488} C_VEL
LIN {X 0,Y 497.003,Z 297.81,A -85,B 0,C 180,E1 5934.763,E2 5934.763} C_VEL
LIN {X 0,Y 497.132,Z 297.81,A -85,B 0,C 180,E1 5939.989,E2 5939.989} C_VEL
LIN {X 0,Y 496.999,Z 297.81,A -85,B 0,C 180,E1 5945.215,E2 5945.215} C_VEL
LIN {X 0,Y 496.858,Z 297.81,A -85,B 0,C 180,E1 5950.489,E2 5950.489} C_VEL
LIN {X 0,Y 496.745,Z 297.81,A -85,B 0,C 180,E1 5955.856,E2 5955.856} C_VEL
LIN {X 0,Y 496.665,Z 297.81,A -85,B 0,C 180,E1 5961.371,E2 5961.371} C_VEL
LIN {X 0,Y 496.451,Z 297.81,A -85,B 0,C 180,E1 5967.114,E2 5967.114} C_VEL
LIN {X 0,Y 496.408,Z 297.81,A -85,B 0,C 180,E1 5973.161,E2 5973.161} C_VEL
LIN {X 0,Y 496.245,Z 297.81,A -85,B 0,C 180,E1 5979.673,E2 5979.673} C_VEL
LIN {X 0,Y 496.334,Z 297.81,A -85,B 0,C 180,E1 5985.822,E2 5985.822} C_VEL
LIN {X 0,Y 492.389,Z 297.81,A -85,B 0,C 180,E1 5987.796,E2 5987.796} C_VEL
LIN {X 0,Y 488.459,Z 297.81,A -85,B 0,C 180,E1 5989.801,E2 5989.801} C_VEL
LIN {X 0,Y 488.468,Z 297.81,A -85,B 0,C 180,E1 5996.215,E2 5996.215} C_VEL
LIN {X 0,Y 488.611,Z 297.81,A -85,B 0,C 180,E1 6002.402,E2 6002.402} C_VEL
LIN {X 0,Y 488.845,Z 297.81,A -85,B 0,C 180,E1 6004.257,E2 6004.257} C_VEL
LIN {X 0,Y 497.073,Z 326.512,A -85,B 0,C 180,E1 6005.055,E2 6005.055} C_VEL
LIN {X 0,Y 496.546,Z 375.275,A -85,B 0,C 180,E1 6005.9,E2 6005.9} C_VEL
LIN {X 0,Y 495.23,Z 408.406,A -85,B 0,C 180,E1 6007.138,E2 6007.138} C_VEL
LIN {X 0,Y 493.634,Z 439.911,A -85,B 0,C 180,E1 6009.057,E2 6009.057} C_VEL
LIN {X 0,Y 492.009,Z 468.625,A -85,B 0,C 180,E1 6011.596,E2 6011.596} C_VEL
LIN {X 0,Y 490.783,Z 493.164,A -85,B 0,C 180,E1 6014.621,E2 6014.621} C_VEL
LIN {X 0,Y 490.08,Z 512.858,A -85,B 0,C 180,E1 6018.004,E2 6018.004} C_VEL
LIN {X 0,Y 489.722,Z 527.237,A -85,B 0,C 180,E1 6021.583,E2 6021.583} C_VEL
LIN {X 0,Y 489.702,Z 535.314,A -85,B 0,C 180,E1 6024.695,E2 6024.695} C_VEL
LIN {X 0,Y 489.718,Z 539.902,A -85,B 0,C 180,E1 6028.234,E2 6028.234} C_VEL
LIN {X 0,Y 489.678,Z 539.857,A -85,B 0,C 180,E1 6031.765,E2 6031.765} C_VEL
LIN {X 0,Y 489.705,Z 535.196,A -85,B 0,C 180,E1 6035.304,E2 6035.304} C_VEL
LIN {X 0,Y 489.78,Z 524.43,A -85,B 0,C 180,E1 6039.177,E2 6039.177} C_VEL
LIN {X 0,Y 490.145,Z 507.889,A -85,B 0,C 180,E1 6042.897,E2 6042.897} C_VEL
LIN {X 0,Y 491.101,Z 486.082,A -85,B 0,C 180,E1 6046.282,E2 6046.282} C_VEL
LIN {X 0,Y 492.385,Z 459.439,A -85,B 0,C 180,E1 6049.238,E2 6049.238} C_VEL
LIN {X 0,Y 494.029,Z 429.059,A -85,B 0,C 180,E1 6051.619,E2 6051.619} C_VEL
LIN {X 0,Y 495.605,Z 396.678,A -85,B 0,C 180,E1 6053.316,E2 6053.316} C_VEL
LIN {X 0,Y 496.635,Z 362.551,A -85,B 0,C 180,E1 6054.346,E2 6054.346} C_VEL
LIN {X 0,Y 496.302,Z 323.284,A -85,B 0,C 180,E1 6054.961,E2 6054.961} C_VEL
LIN {X 0,Y 488.728,Z 297.81,A -85,B 0,C 180,E1 6055.712,E2 6055.712} C_VEL
LIN {X 0,Y 488.493,Z 297.81,A -85,B 0,C 180,E1 6061.677,E2 6061.677} C_VEL
LIN {X 0,Y 488.294,Z 297.81,A -85,B 0,C 180,E1 6068.175,E2 6068.175} C_VEL
LIN {X 0,Y 488.353,Z 297.81,A -85,B 0,C 180,E1 6074.722,E2 6074.722} C_VEL
LIN {X 0,Y 488.42,Z 297.81,A -85,B 0,C 180,E1 6080.568,E2 6080.568} C_VEL
LIN {X 0,Y 488.422,Z 297.81,A -85,B 0,C 180,E1 6086.529,E2 6086.529} C_VEL
LIN {X 0,Y 488.513,Z 297.81,A -85,B 0,C 180,E1 6092.408,E2 6092.408} C_VEL
LIN {X 0,Y 488.659,Z 297.81,A -85,B 0,C 180,E1 6098.261,E2 6098.261} C_VEL
LIN {X 0,Y 488.706,Z 297.81,A -85,B 0,C 180,E1 6103.876,E2 6103.876} C_VEL
LIN {X 0,Y 488.811,Z 297.81,A -85,B 0,C 180,E1 6109.337,E2 6109.337} C_VEL
LIN {X 0,Y 489.098,Z 297.81,A -85,B 0,C 180,E1 6114.7,E2 6114.7} C_VEL
LIN {X 0,Y 489.148,Z 297.81,A -85,B 0,C 180,E1 6120.011,E2 6120.011} C_VEL
LIN {X 0,Y 489.042,Z 297.81,A -85,B 0,C 180,E1 6125.323,E2 6125.323} C_VEL
LIN {X 0,Y 488.893,Z 297.81,A -85,B 0,C 180,E1 6130.684,E2 6130.684} C_VEL
LIN {X 0,Y 488.783,Z 297.81,A -85,B 0,C 180,E1 6136.856,E2 6136.856} C_VEL
LIN {X 0,Y 488.668,Z 297.81,A -85,B 0,C 180,E1 6142.122,E2 6142.122} C_VEL
LIN {X 0,Y 488.529,Z 297.81,A -85,B 0,C 180,E1 6147.616,E2 6147.616} C_VEL
LIN {X 0,Y 488.77,Z 297.81,A -85,B 0,C 180,E1 6154.176,E2 6154.176} C_VEL
LIN {X 0,Y 494.039,Z 320.75,A -85,B 0,C 180,E1 6155.304,E2 6155.304} C_VEL
LIN {X 0,Y 493.125,Z 345.33,A -85,B 0,C 180,E1 6156.878,E2 6156.878} C_VEL
LIN {X 0,Y 492.033,Z 366.156,A -85,B 0,C 180,E1 6158.948,E2 6158.948} C_VEL
LIN {X 0,Y 491.089,Z 383.202,A -85,B 0,C 180,E1 6161.518,E2 6161.518} C_VEL
LIN {X 0,Y 490.526,Z 395.782,A -85,B 0,C 180,E1 6164.58,E2 6164.58} C_VEL
LIN {X 0,Y 490.073,Z 402.241,A -85,B 0,C 180,E1 6167.664,E2 6167.664} C_VEL
LIN {X 0,Y 489.913,Z 403.476,A -85,B 0,C 180,E1 6170.376,E2 6170.376} C_VEL
LIN {X 0,Y 490.151,Z 399.493,A -85,B 0,C 180,E1 6173.704,E2 6173.704} C_VEL
LIN {X 0,Y 490.654,Z 389.597,A -85,B 0,C 180,E1 6176.868,E2 6176.868} C_VEL
LIN {X 0,Y 491.411,Z 374.537,A -85,B 0,C 180,E1 6179.66,E2 6179.66} C_VEL
LIN {X 0,Y 492.341,Z 354.486,A -85,B 0,C 180,E1 6182.063,E2 6182.063} C_VEL
LIN {X 0,Y 493.288,Z 330.496,A -85,B 0,C 180,E1 6183.924,E2 6183.924} C_VEL
LIN {X 0,Y 492.72,Z 313.413,A -85,B 0,C 180,E1 6184.837,E2 6184.837} C_VEL
LIN {X 0,Y 488.864,Z 297.81,A -85,B 0,C 180,E1 6185.565,E2 6185.565} C_VEL
LIN {X 0,Y 488.855,Z 297.81,A -85,B 0,C 180,E1 6192.021,E2 6192.021} C_VEL
LIN {X 0,Y 488.712,Z 297.81,A -85,B 0,C 180,E1 6197.518,E2 6197.518} C_VEL
LIN {X 0,Y 488.951,Z 298.181,A -85,B 0,C 180,E1 6200.788,E2 6200.788} C_VEL
LIN {X 0,Y 493.09,Z 321.118,A -85,B 0,C 180,E1 6201.698,E2 6201.698} C_VEL
LIN {X 0,Y 492.484,Z 345.445,A -85,B 0,C 180,E1 6203.182,E2 6203.182} C_VEL
LIN {X 0,Y 491.654,Z 365.887,A -85,B 0,C 180,E1 6205.159,E2 6205.159} C_VEL
LIN {X 0,Y 490.961,Z 382.405,A -85,B 0,C 180,E1 6207.578,E2 6207.578} C_VEL
LIN {X 0,Y 490.418,Z 395.043,A -85,B 0,C 180,E1 6210.54,E2 6210.54} C_VEL
LIN {X 0,Y 490.123,Z 401.732,A -85,B 0,C 180,E1 6213.531,E2 6213.531} C_VEL
LIN {X 0,Y 490.026,Z 403.287,A -85,B 0,C 180,E1 6215.301,E2 6215.301} C_VEL
LIN {X 0,Y 489.996,Z 403.07,A -85,B 0,C 180,E1 6217.076,E2 6217.076} C_VEL
LIN {X 0,Y 490.289,Z 399.138,A -85,B 0,C 180,E1 6219.9,E2 6219.9} C_VEL
LIN {X 0,Y 490.661,Z 389.662,A -85,B 0,C 180,E1 6222.884,E2 6222.884} C_VEL
LIN {X 0,Y 491.37,Z 375.072,A -85,B 0,C 180,E1 6225.588,E2 6225.588} C_VEL
LIN {X 0,Y 492.13,Z 356.222,A -85,B 0,C 180,E1 6227.857,E2 6227.857} C_VEL
LIN {X 0,Y 493.017,Z 332.527,A -85,B 0,C 180,E1 6229.675,E2 6229.675} C_VEL
LIN {X 0,Y 492.367,Z 313.012,A -85,B 0,C 180,E1 6230.643,E2 6230.643} C_VEL
LIN {X 0,Y 488.83,Z 297.81,A -85,B 0,C 180,E1 6231.27,E2 6231.27} C_VEL
LIN {X 0,Y 488.469,Z 297.81,A -85,B 0,C 180,E1 6237.606,E2 6237.606} C_VEL
LIN {X 0,Y 488.45,Z 297.81,A -85,B 0,C 180,E1 6243.786,E2 6243.786} C_VEL
LIN {X 0,Y 488.42,Z 297.81,A -85,B 0,C 180,E1 6249.412,E2 6249.412} C_VEL
LIN {X 0,Y 488.381,Z 297.81,A -85,B 0,C 180,E1 6255.289,E2 6255.289} C_VEL
LIN {X 0,Y 488.43,Z 297.81,A -85,B 0,C 180,E1 6261.822,E2 6261.822} C_VEL
LIN {X 0,Y 488.408,Z 297.81,A -85,B 0,C 180,E1 6268.302,E2 6268.302} C_VEL
LIN {X 0,Y 488.538,Z 297.81,A -85,B 0,C 180,E1 6274.365,E2 6274.365} C_VEL
LIN {X 0,Y 488.825,Z 297.81,A -85,B 0,C 180,E1 6280.137,E2 6280.137} C_VEL
LIN {X 0,Y 488.679,Z 297.81,A -85,B 0,C 180,E1 6285.686,E2 6285.686} C_VEL
LIN {X 0,Y 488.932,Z 297.81,A -85,B 0,C 180,E1 6291.111,E2 6291.111} C_VEL
LIN {X 0,Y 489.074,Z 297.81,A -85,B 0,C 180,E1 6296.451,E2 6296.451} C_VEL
LIN {X 0,Y 489.092,Z 297.81,A -85,B 0,C 180,E1 6301.757,E2 6301.757} C_VEL
LIN {X 0,Y 488.994,Z 297.81,A -85,B 0,C 180,E1 6307.08,E2 6307.08} C_VEL
LIN {X 0,Y 488.925,Z 297.81,A -85,B 0,C 180,E1 6312.466,E2 6312.466} C_VEL
LIN {X 0,Y 488.792,Z 297.81,A -85,B 0,C 180,E1 6317.971,E2 6317.971} C_VEL
LIN {X 0,Y 488.669,Z 297.81,A -85,B 0,C 180,E1 6323.657,E2 6323.657} C_VEL
LIN {X 0,Y 488.452,Z 297.81,A -85,B 0,C 180,E1 6330.115,E2 6330.115} C_VEL
LIN {X 0,Y 488.36,Z 297.81,A -85,B 0,C 180,E1 6335.938,E2 6335.938} C_VEL
LIN {X 0,Y 488.357,Z 297.81,A -85,B 0,C 180,E1 6342.133,E2 6342.133} C_VEL
LIN {X 0,Y 488.449,Z 297.81,A -85,B 0,C 180,E1 6347.84,E2 6347.84} C_VEL
LIN {X 0,Y 488.459,Z 297.81,A -85,B 0,C 180,E1 6349.801,E2 6349.801} C_VEL
LIN {X 0,Y 487.204,Z 297.81,A -85,B 0,C 180,E1 6350.815,E2 6350.815} C_VEL
LIN {X 0,Y 480.524,Z 297.81,A -85,B 0,C 180,E1 6353.843,E2 6353.843} C_VEL
LIN {X 0,Y 480.601,Z 297.81,A -85,B 0,C 180,E1 6359.843,E2 6359.843} C_VEL
LIN {X 0,Y 480.89,Z 297.81,A -85,B 0,C 180,E1 6363.89,E2 6363.89} C_VEL
LIN {X 0,Y 489.648,Z 328.652,A -85,B 0,C 180,E1 6364.767,E2 6364.767} C_VEL
LIN {X 0,Y 489.131,Z 374.549,A -85,B 0,C 180,E1 6365.58,E2 6365.58} C_VEL
LIN {X 0,Y 487.737,Z 407.573,A -85,B 0,C 180,E1 6366.827,E2 6366.827} C_VEL
LIN {X 0,Y 485.979,Z 438.973,A -85,B 0,C 180,E1 6368.761,E2 6368.761} C_VEL
LIN {X 0,Y 484.22,Z 468.02,A -85,B 0,C 180,E1 6371.371,E2 6371.371} C_VEL
LIN {X 0,Y 482.897,Z 493.451,A -85,B 0,C 180,E1 6374.596,E2 6374.596} C_VEL
LIN {X 0,Y 482.201,Z 512.818,A -85,B 0,C 180,E1 6378.034,E2 6378.034} C_VEL
LIN {X 0,Y 481.873,Z 527.522,A -85,B 0,C 180,E1 6381.898,E2 6381.898} C_VEL
LIN {X 0,Y 481.834,Z 535.844,A -85,B 0,C 180,E1 6385.509,E2 6385.509} C_VEL
LIN {X 0,Y 481.889,Z 538.816,A -85,B 0,C 180,E1 6388.205,E2 6388.205} C_VEL
LIN {X 0,Y 481.858,Z 538.762,A -85,B 0,C 180,E1 6391.794,E2 6391.794} C_VEL
LIN {X 0,Y 481.876,Z 534.075,A -85,B 0,C 180,E1 6395.39,E2 6395.39} C_VEL
LIN {X 0,Y 481.899,Z 524.397,A -85,B 0,C 180,E1 6399.007,E2 6399.007} C_VEL
LIN {X 0,Y 482.197,Z 508.996,A -85,B 0,C 180,E1 6402.653,E2 6402.653} C_VEL
LIN {X 0,Y 483.123,Z 488.086,A -85,B 0,C 180,E1 6406.093,E2 6406.093} C_VEL
LIN {X 0,Y 484.429,Z 462.773,A -85,B 0,C 180,E1 6409.091,E2 6409.091} C_VEL
LIN {X 0,Y 486.235,Z 432.628,A -85,B 0,C 180,E1 6411.619,E2 6411.619} C_VEL
LIN {X 0,Y 487.869,Z 401.051,A -85,B 0,C 180,E1 6413.407,E2 6413.407} C_VEL
LIN {X 0,Y 489.11,Z 367.849,A -85,B 0,C 180,E1 6414.536,E2 6414.536} C_VEL
LIN {X 0,Y 488.795,Z 324.423,A -85,B 0,C 180,E1 6415.272,E2 6415.272} C_VEL
LIN {X 0,Y 480.774,Z 297.81,A -85,B 0,C 180,E1 6416.066,E2 6416.066} C_VEL
LIN {X 0,Y 480.566,Z 297.81,A -85,B 0,C 180,E1 6422.262,E2 6422.262} C_VEL
LIN {X 0,Y 480.366,Z 297.81,A -85,B 0,C 180,E1 6428.922,E2 6428.922} C_VEL
LIN {X 0,Y 480.362,Z 297.81,A -85,B 0,C 180,E1 6433.752,E2 6433.752} C_VEL
LIN {X 0,Y 480.466,Z 297.81,A -85,B 0,C 180,E1 6438.917,E2 6438.917} C_VEL
LIN {X 0,Y 480.453,Z 297.81,A -85,B 0,C 180,E1 6444.745,E2 6444.745} C_VEL
LIN {X 0,Y 480.502,Z 297.81,A -85,B 0,C 180,E1 6449.848,E2 6449.848} C_VEL
LIN {X 0,Y 480.647,Z 297.81,A -85,B 0,C 180,E1 6455.924,E2 6455.924} C_VEL
LIN {X 0,Y 480.859,Z 297.81,A -85,B 0,C 180,E1 6461.722,E2 6461.722} C_VEL
LIN {X 0,Y 480.761,Z 297.81,A -85,B 0,C 180,E1 6467.319,E2 6467.319} C_VEL
LIN {X 0,Y 481.102,Z 297.81,A -85,B 0,C 180,E1 6472.804,E2 6472.804} C_VEL
LIN {X 0,Y 481.414,Z 297.81,A -85,B 0,C 180,E1 6478.215,E2 6478.215} C_VEL
LIN {X 0,Y 481.245,Z 297.81,A -85,B 0,C 180,E1 6483.607,E2 6483.607} C_VEL
LIN {X 0,Y 481.075,Z 297.81,A -85,B 0,C 180,E1 6489.035,E2 6489.035} C_VEL
LIN {X 0,Y 480.965,Z 297.81,A -85,B 0,C 180,E1 6494.548,E2 6494.548} C_VEL
LIN {X 0,Y 480.804,Z 297.81,A -85,B 0,C 180,E1 6500.209,E2 6500.209} C_VEL
LIN {X 0,Y 480.647,Z 297.81,A -85,B 0,C 180,E1 6506.087,E2 6506.087} C_VEL
LIN {X 0,Y 480.762,Z 297.81,A -85,B 0,C 180,E1 6513.167,E2 6513.167} C_VEL
LIN {X 0,Y 480.879,Z 298.334,A -85,B 0,C 180,E1 6513.842,E2 6513.842} C_VEL
LIN {X 0,Y 486.561,Z 322.807,A -85,B 0,C 180,E1 6515.077,E2 6515.077} C_VEL
LIN {X 0,Y 485.471,Z 348.467,A -85,B 0,C 180,E1 6516.807,E2 6516.807} C_VEL
LIN {X 0,Y 484.341,Z 369.049,A -85,B 0,C 180,E1 6518.976,E2 6518.976} C_VEL
LIN {X 0,Y 483.348,Z 384.887,A -85,B 0,C 180,E1 6521.473,E2 6521.473} C_VEL
LIN {X 0,Y 482.823,Z 395.525,A -85,B 0,C 180,E1 6524.043,E2 6524.043} C_VEL
LIN {X 0,Y 482.443,Z 401.728,A -85,B 0,C 180,E1 6526.519,E2 6526.519} C_VEL
LIN {X 0,Y 482.146,Z 404.418,A -85,B 0,C 180,E1 6528.91,E2 6528.91} C_VEL
LIN {X 0,Y 482.211,Z 402.79,A -85,B 0,C 180,E1 6532.494,E2 6532.494} C_VEL
LIN {X 0,Y 482.709,Z 395.177,A -85,B 0,C 180,E1 6535.758,E2 6535.758} C_VEL
LIN {X 0,Y 483.333,Z 382.62,A -85,B 0,C 180,E1 6538.652,E2 6538.652} C_VEL
LIN {X 0,Y 484.284,Z 364.267,A -85,B 0,C 180,E1 6541.325,E2 6541.325} C_VEL
LIN {X 0,Y 485.319,Z 342.561,A -85,B 0,C 180,E1 6543.4,E2 6543.4} C_VEL
LIN {X 0,Y 485.578,Z 316.604,A -85,B 0,C 180,E1 6544.986,E2 6544.986} C_VEL
LIN {X 0,Y 480.924,Z 297.81,A -85,B 0,C 180,E1 6545.928,E2 6545.928} C_VEL
LIN {X 0,Y 480.915,Z 297.81,A -85,B 0,C 180,E1 6551.714,E2 6551.714} C_VEL
LIN {X 0,Y 480.783,Z 297.81,A -85,B 0,C 180,E1 6557.309,E2 6557.309} C_VEL
LIN {X 0,Y 481.028,Z 297.829,A -85,B 0,C 180,E1 6560.523,E2 6560.523} C_VEL
LIN {X 0,Y 485.462,Z 321.942,A -85,B 0,C 180,E1 6561.477,E2 6561.477} C_VEL
LIN {X 0,Y 484.852,Z 346.084,A -85,B 0,C 180,E1 6562.961,E2 6562.961} C_VEL
LIN {X 0,Y 483.946,Z 367.597,A -85,B 0,C 180,E1 6565.081,E2 6565.081} C_VEL
LIN {X 0,Y 483.203,Z 383.915,A -85,B 0,C 180,E1 6567.539,E2 6567.539} C_VEL
LIN {X 0,Y 482.64,Z 396.055,A -85,B 0,C 180,E1 6570.448,E2 6570.448} C_VEL
LIN {X 0,Y 482.317,Z 402.914,A -85,B 0,C 180,E1 6573.588,E2 6573.588} C_VEL
LIN {X 0,Y 482.217,Z 404.384,A -85,B 0,C 180,E1 6575.387,E2 6575.387} C_VEL
LIN {X 0,Y 482.242,Z 403.323,A -85,B 0,C 180,E1 6578.095,E2 6578.095} C_VEL
LIN {X 0,Y 482.674,Z 396.915,A -85,B 0,C 180,E1 6581.268,E2 6581.268} C_VEL
LIN {X 0,Y 483.168,Z 384.992,A -85,B 0,C 180,E1 6584.253,E2 6584.253} C_VEL
LIN {X 0,Y 484.019,Z 368.904,A -85,B 0,C 180,E1 6586.762,E2 6586.762} C_VEL
LIN {X 0,Y 484.957,Z 347.984,A -85,B 0,C 180,E1 6588.896,E2 6588.896} C_VEL
LIN {X 0,Y 485.717,Z 323.041,A -85,B 0,C 180,E1 6590.477,E2 6590.477} C_VEL
LIN {X 0,Y 481.954,Z 302.493,A -85,B 0,C 180,E1 6591.375,E2 6591.375} C_VEL
LIN {X 0,Y 480.883,Z 297.81,A -85,B 0,C 180,E1 6591.547,E2 6591.547} C_VEL
LIN {X 0,Y 480.483,Z 297.81,A -85,B 0,C 180,E1 6598.407,E2 6598.407} C_VEL
LIN {X 0,Y 480.478,Z 297.81,A -85,B 0,C 180,E1 6604.424,E2 6604.424} C_VEL
LIN {X 0,Y 480.522,Z 297.81,A -85,B 0,C 180,E1 6608.908,E2 6608.908} C_VEL
LIN {X 0,Y 480.407,Z 297.81,A -85,B 0,C 180,E1 6613.725,E2 6613.725} C_VEL
LIN {X 0,Y 480.491,Z 297.81,A -85,B 0,C 180,E1 6618.915,E2 6618.915} C_VEL
LIN {X 0,Y 480.438,Z 297.81,A -85,B 0,C 180,E1 6624.749,E2 6624.749} C_VEL
LIN {X 0,Y 480.49,Z 297.81,A -85,B 0,C 180,E1 6629.821,E2 6629.821} C_VEL
LIN {X 0,Y 480.637,Z 297.81,A -85,B 0,C 180,E1 6635.899,E2 6635.899} C_VEL
LIN {X 0,Y 480.921,Z 297.81,A -85,B 0,C 180,E1 6641.701,E2 6641.701} C_VEL
LIN {X 0,Y 480.822,Z 297.81,A -85,B 0,C 180,E1 6647.298,E2 6647.298} C_VEL
LIN {X 0,Y 481.133,Z 297.81,A -85,B 0,C 180,E1 6652.992,E2 6652.992} C_VEL
LIN {X 0,Y 481.427,Z 297.81,A -85,B 0,C 180,E1 6658.193,E2 6658.193} C_VEL
LIN {X 0,Y 481.301,Z 297.81,A -85,B 0,C 180,E1 6663.584,E2 6663.584} C_VEL
LIN {X 0,Y 481.086,Z 297.81,A -85,B 0,C 180,E1 6669.012,E2 6669.012} C_VEL
LIN {X 0,Y 480.962,Z 297.81,A -85,B 0,C 180,E1 6674.525,E2 6674.525} C_VEL
LIN {X 0,Y 480.825,Z 297.81,A -85,B 0,C 180,E1 6680.184,E2 6680.184} C_VEL
LIN {X 0,Y 480.649,Z 297.81,A -85,B 0,C 180,E1 6686.062,E2 6686.062} C_VEL
LIN {X 0,Y 480.526,Z 297.81,A -85,B 0,C 180,E1 6692.254,E2 6692.254} C_VEL
LIN {X 0,Y 480.425,Z 297.81,A -85,B 0,C 180,E1 6698.904,E2 6698.904} C_VEL
LIN {X 0,Y 480.423,Z 297.81,A -85,B 0,C 180,E1 6703.744,E2 6703.744} C_VEL
LIN {X 0,Y 480.465,Z 297.81,A -85,B 0,C 180,E1 6709.799,E2 6709.799} C_VEL
LIN {X 0,Y 480.524,Z 297.81,A -85,B 0,C 180,E1 6713.843,E2 6713.843} C_VEL
LIN {X 0,Y 479.216,Z 297.81,A -85,B 0,C 180,E1 6714.876,E2 6714.876} C_VEL
LIN {X 0,Y 472.611,Z 297.81,A -85,B 0,C 180,E1 6717.692,E2 6717.692} C_VEL
LIN {X 0,Y 472.519,Z 297.81,A -85,B 0,C 180,E1 6717.959,E2 6717.959} C_VEL
LIN {X 0,Y 472.931,Z 297.93,A -85,B 0,C 180,E1 6723.545,E2 6723.545} C_VEL
LIN {X 0,Y 482.233,Z 330.172,A -85,B 0,C 180,E1 6724.463,E2 6724.463} C_VEL
LIN {X 0,Y 481.653,Z 375.022,A -85,B 0,C 180,E1 6725.284,E2 6725.284} C_VEL
LIN {X 0,Y 480.146,Z 407.811,A -85,B 0,C 180,E1 6726.561,E2 6726.561} C_VEL
LIN {X 0,Y 478.287,Z 439.459,A -85,B 0,C 180,E1 6728.564,E2 6728.564} C_VEL
LIN {X 0,Y 476.467,Z 467.735,A -85,B 0,C 180,E1 6731.177,E2 6731.177} C_VEL
LIN {X 0,Y 475.062,Z 492.216,A -85,B 0,C 180,E1 6734.335,E2 6734.335} C_VEL
LIN {X 0,Y 474.311,Z 511.647,A -85,B 0,C 180,E1 6737.832,E2 6737.832} C_VEL
LIN {X 0,Y 473.998,Z 526.406,A -85,B 0,C 180,E1 6741.763,E2 6741.763} C_VEL
LIN {X 0,Y 473.989,Z 534.751,A -85,B 0,C 180,E1 6745.434,E2 6745.434} C_VEL
LIN {X 0,Y 474.063,Z 537.73,A -85,B 0,C 180,E1 6748.175,E2 6748.175} C_VEL
LIN {X 0,Y 474.034,Z 537.667,A -85,B 0,C 180,E1 6751.824,E2 6751.824} C_VEL
LIN {X 0,Y 474.051,Z 532.955,A -85,B 0,C 180,E1 6755.479,E2 6755.479} C_VEL
LIN {X 0,Y 474.061,Z 522.41,A -85,B 0,C 180,E1 6759.39,E2 6759.39} C_VEL
LIN {X 0,Y 474.359,Z 507.766,A -85,B 0,C 180,E1 6762.866,E2 6762.866} C_VEL
LIN {X 0,Y 475.335,Z 486.762,A -85,B 0,C 180,E1 6766.364,E2 6766.364} C_VEL
LIN {X 0,Y 476.731,Z 461.301,A -85,B 0,C 180,E1 6769.411,E2 6769.411} C_VEL
LIN {X 0,Y 478.644,Z 431.046,A -85,B 0,C 180,E1 6771.974,E2 6771.974} C_VEL
LIN {X 0,Y 480.455,Z 398.954,A -85,B 0,C 180,E1 6773.79,E2 6773.79} C_VEL
LIN {X 0,Y 481.721,Z 365.666,A -85,B 0,C 180,E1 6774.905,E2 6774.905} C_VEL
LIN {X 0,Y 481.25,Z 325.233,A -85,B 0,C 180,E1 6775.603,E2 6775.603} C_VEL
LIN {X 0,Y 472.795,Z 297.81,A -85,B 0,C 180,E1 6776.466,E2 6776.466} C_VEL
LIN {X 0,Y 472.564,Z 297.81,A -85,B 0,C 180,E1 6782.877,E2 6782.877} C_VEL
LIN {X 0,Y 472.504,Z 297.81,A -85,B 0,C 180,E1 6787.357,E2 6787.357} C_VEL
LIN {X 0,Y 472.401,Z 297.81,A -85,B 0,C 180,E1 6794.647,E2 6794.647} C_VEL
LIN {X 0,Y 472.522,Z 297.81,A -85,B 0,C 180,E1 6800.318,E2 6800.318} C_VEL
LIN {X 0,Y 472.499,Z 297.81,A -85,B 0,C 180,E1 6806.134,E2 6806.134} C_VEL
LIN {X 0,Y 472.623,Z 297.81,A -85,B 0,C 180,E1 6811.397,E2 6811.397} C_VEL
LIN {X 0,Y 472.827,Z 297.81,A -85,B 0,C 180,E1 6817.745,E2 6817.745} C_VEL
LIN {X 0,Y 472.89,Z 297.81,A -85,B 0,C 180,E1 6823.322,E2 6823.322} C_VEL
LIN {X 0,Y 472.943,Z 297.81,A -85,B 0,C 180,E1 6828.974,E2 6828.974} C_VEL
LIN {X 0,Y 473.268,Z 297.81,A -85,B 0,C 180,E1 6834.522,E2 6834.522} C_VEL
LIN {X 0,Y 473.354,Z 297.81,A -85,B 0,C 180,E1 6840.011,E2 6840.011} C_VEL
LIN {X 0,Y 473.214,Z 297.81,A -85,B 0,C 180,E1 6845.501,E2 6845.501} C_VEL
LIN {X 0,Y 473.048,Z 297.81,A -85,B 0,C 180,E1 6851.046,E2 6851.046} C_VEL
LIN {X 0,Y 472.949,Z 297.81,A -85,B 0,C 180,E1 6856.829,E2 6856.829} C_VEL
LIN {X 0,Y 472.826,Z 297.81,A -85,B 0,C 180,E1 6862.531,E2 6862.531} C_VEL
LIN {X 0,Y 472.676,Z 297.81,A -85,B 0,C 180,E1 6868.625,E2 6868.625} C_VEL
LIN {X 0,Y 472.889,Z 297.833,A -85,B 0,C 180,E1 6873.447,E2 6873.447} C_VEL
LIN {X 0,Y 479.122,Z 323.881,A -85,B 0,C 180,E1 6874.793,E2 6874.793} C_VEL
LIN {X 0,Y 477.948,Z 349.486,A -85,B 0,C 180,E1 6876.553,E2 6876.553} C_VEL
LIN {X 0,Y 476.679,Z 371.089,A -85,B 0,C 180,E1 6878.897,E2 6878.897} C_VEL
LIN {X 0,Y 475.613,Z 386.675,A -85,B 0,C 180,E1 6881.447,E2 6881.447} C_VEL
LIN {X 0,Y 474.971,Z 397.97,A -85,B 0,C 180,E1 6884.36,E2 6884.36} C_VEL
LIN {X 0,Y 474.543,Z 403.763,A -85,B 0,C 180,E1 6887.021,E2 6887.021} C_VEL
LIN {X 0,Y 474.281,Z 405.639,A -85,B 0,C 180,E1 6890.482,E2 6890.482} C_VEL
LIN {X 0,Y 474.544,Z 401.803,A -85,B 0,C 180,E1 6893.75,E2 6893.75} C_VEL
LIN {X 0,Y 475.102,Z 392.389,A -85,B 0,C 180,E1 6896.922,E2 6896.922} C_VEL
LIN {X 0,Y 475.922,Z 378.229,A -85,B 0,C 180,E1 6899.733,E2 6899.733} C_VEL
LIN {X 0,Y 476.989,Z 359.039,A -85,B 0,C 180,E1 6902.22,E2 6902.22} C_VEL
LIN {X 0,Y 478.118,Z 334.968,A -85,B 0,C 180,E1 6904.249,E2 6904.249} C_VEL
LIN {X 0,Y 477.747,Z 316.796,A -85,B 0,C 180,E1 6905.303,E2 6905.303} C_VEL
LIN {X 0,Y 472.977,Z 297.81,A -85,B 0,C 180,E1 6906.248,E2 6906.248} C_VEL
LIN {X 0,Y 472.992,Z 297.81,A -85,B 0,C 180,E1 6911.396,E2 6911.396} C_VEL
LIN {X 0,Y 472.877,Z 297.81,A -85,B 0,C 180,E1 6917.093,E2 6917.093} C_VEL
LIN {X 0,Y 473.144,Z 297.81,A -85,B 0,C 180,E1 6920.251,E2 6920.251} C_VEL
LIN {X 0,Y 477.806,Z 323.647,A -85,B 0,C 180,E1 6921.291,E2 6921.291} C_VEL
LIN {X 0,Y 477.14,Z 348.131,A -85,B 0,C 180,E1 6922.847,E2 6922.847} C_VEL
LIN {X 0,Y 476.218,Z 369.287,A -85,B 0,C 180,E1 6925.001,E2 6925.001} C_VEL
LIN {X 0,Y 475.36,Z 386.529,A -85,B 0,C 180,E1 6927.726,E2 6927.726} C_VEL
LIN {X 0,Y 474.833,Z 397.387,A -85,B 0,C 180,E1 6930.456,E2 6930.456} C_VEL
LIN {X 0,Y 474.485,Z 404.096,A -85,B 0,C 180,E1 6933.647,E2 6933.647} C_VEL
LIN {X 0,Y 474.383,Z 405.48,A -85,B 0,C 180,E1 6935.477,E2 6935.477} C_VEL
LIN {X 0,Y 474.439,Z 404.302,A -85,B 0,C 180,E1 6938.229,E2 6938.229} C_VEL
LIN {X 0,Y 474.92,Z 397.766,A -85,B 0,C 180,E1 6941.455,E2 6941.455} C_VEL
LIN {X 0,Y 475.493,Z 385.671,A -85,B 0,C 180,E1 6944.488,E2 6944.488} C_VEL
LIN {X 0,Y 476.467,Z 367.906,A -85,B 0,C 180,E1 6947.22,E2 6947.22} C_VEL
LIN {X 0,Y 477.535,Z 345.871,A -85,B 0,C 180,E1 6949.378,E2 6949.378} C_VEL
LIN {X 0,Y 478.18,Z 321.281,A -85,B 0,C 180,E1 6950.863,E2 6950.863} C_VEL
LIN {X 0,Y 472.942,Z 297.81,A -85,B 0,C 180,E1 6951.929,E2 6951.929} C_VEL
LIN {X 0,Y 472.571,Z 297.81,A -85,B 0,C 180,E1 6958.619,E2 6958.619} C_VEL
LIN {X 0,Y 472.605,Z 297.81,A -85,B 0,C 180,E1 6965.081,E2 6965.081} C_VEL
LIN {X 0,Y 472.518,Z 297.81,A -85,B 0,C 180,E1 6969.944,E2 6969.944} C_VEL
LIN {X 0,Y 472.456,Z 297.81,A -85,B 0,C 180,E1 6975.341,E2 6975.341} C_VEL
LIN {X 0,Y 472.526,Z 297.81,A -85,B 0,C 180,E1 6980.289,E2 6980.289} C_VEL
LIN {X 0,Y 472.502,Z 297.81,A -85,B 0,C 180,E1 6986.135,E2 6986.135} C_VEL
LIN {X 0,Y 472.584,Z 297.81,A -85,B 0,C 180,E1 6991.368,E2 6991.368} C_VEL
LIN {X 0,Y 472.867,Z 297.81,A -85,B 0,C 180,E1 6997.736,E2 6997.736} C_VEL
LIN {X 0,Y 472.957,Z 297.81,A -85,B 0,C 180,E1 7003.3,E2 7003.3} C_VEL
LIN {X 0,Y 473.001,Z 297.81,A -85,B 0,C 180,E1 7008.953,E2 7008.953} C_VEL
LIN {X 0,Y 473.266,Z 297.81,A -85,B 0,C 180,E1 7014.499,E2 7014.499} C_VEL
LIN {X 0,Y 473.452,Z 297.81,A -85,B 0,C 180,E1 7019.989,E2 7019.989} C_VEL
LIN {X 0,Y 473.251,Z 297.81,A -85,B 0,C 180,E1 7025.478,E2 7025.478} C_VEL
LIN {X 0,Y 473.106,Z 297.81,A -85,B 0,C 180,E1 7031.022,E2 7031.022} C_VEL
LIN {X 0,Y 472.941,Z 297.81,A -85,B 0,C 180,E1 7036.822,E2 7036.822} C_VEL
LIN {X 0,Y 472.854,Z 297.81,A -85,B 0,C 180,E1 7042.505,E2 7042.505} C_VEL
LIN {X 0,Y 472.651,Z 297.81,A -85,B 0,C 180,E1 7048.601,E2 7048.601} C_VEL
LIN {X 0,Y 472.563,Z 297.81,A -85,B 0,C 180,E1 7055.072,E2 7055.072} C_VEL
LIN {X 0,Y 472.431,Z 297.81,A -85,B 0,C 180,E1 7059.951,E2 7059.951} C_VEL
LIN {X 0,Y 472.472,Z 297.81,A -85,B 0,C 180,E1 7065.36,E2 7065.36} C_VEL
LIN {X 0,Y 472.577,Z 297.81,A -85,B 0,C 180,E1 7070.31,E2 7070.31} C_VEL
LIN {X 0,Y 472.562,Z 297.81,A -85,B 0,C 180,E1 7076.105,E2 7076.105} C_VEL
LIN {X 0,Y 472.519,Z 297.81,A -85,B 0,C 180,E1 7077.959,E2 7077.959} C_VEL
LIN {X 0,Y 471.286,Z 297.81,A -85,B 0,C 180,E1 7079.007,E2 7079.007} C_VEL
LIN {X 0,Y 464.896,Z 297.81,A -85,B 0,C 180,E1 7081.869,E2 7081.869} C_VEL
LIN {X 0,Y 464.826,Z 297.81,A -85,B 0,C 180,E1 7082.14,E2 7082.14} C_VEL
LIN {X 0,Y 465.005,Z 298.268,A -85,B 0,C 180,E1 7083.17,E2 7083.17} C_VEL
LIN {X 0,Y 474.779,Z 329.367,A -85,B 0,C 180,E1 7084.112,E2 7084.112} C_VEL
LIN {X 0,Y 474.244,Z 374.226,A -85,B 0,C 180,E1 7084.945,E2 7084.945} C_VEL
LIN {X 0,Y 472.579,Z 407.986,A -85,B 0,C 180,E1 7086.288,E2 7086.288} C_VEL
LIN {X 0,Y 470.666,Z 438.657,A -85,B 0,C 180,E1 7088.266,E2 7088.266} C_VEL
LIN {X 0,Y 468.694,Z 467.43,A -85,B 0,C 180,E1 7090.974,E2 7090.974} C_VEL
LIN {X 0,Y 467.28,Z 490.967,A -85,B 0,C 180,E1 7094.068,E2 7094.068} C_VEL
LIN {X 0,Y 466.392,Z 510.464,A -85,B 0,C 180,E1 7097.622,E2 7097.622} C_VEL
LIN {X 0,Y 466.126,Z 525.304,A -85,B 0,C 180,E1 7101.63,E2 7101.63} C_VEL
LIN {X 0,Y 466.144,Z 533.655,A -85,B 0,C 180,E1 7105.357,E2 7105.357} C_VEL
LIN {X 0,Y 466.246,Z 536.643,A -85,B 0,C 180,E1 7108.145,E2 7108.145} C_VEL
LIN {X 0,Y 466.222,Z 536.572,A -85,B 0,C 180,E1 7111.854,E2 7111.854} C_VEL
LIN {X 0,Y 466.217,Z 531.833,A -85,B 0,C 180,E1 7115.572,E2 7115.572} C_VEL
LIN {X 0,Y 466.203,Z 521.237,A -85,B 0,C 180,E1 7119.549,E2 7119.549} C_VEL
LIN {X 0,Y 466.594,Z 505.231,A -85,B 0,C 180,E1 7123.354,E2 7123.354} C_VEL
LIN {X 0,Y 467.643,Z 483.775,A -85,B 0,C 180,E1 7126.882,E2 7126.882} C_VEL
LIN {X 0,Y 469.288,Z 457.48,A -85,B 0,C 180,E1 7129.977,E2 7129.977} C_VEL
LIN {X 0,Y 471.184,Z 428.063,A -85,B 0,C 180,E1 7132.431,E2 7132.431} C_VEL
LIN {X 0,Y 473.089,Z 395.576,A -85,B 0,C 180,E1 7134.246,E2 7134.246} C_VEL
LIN {X 0,Y 474.46,Z 361.426,A -85,B 0,C 180,E1 7135.331,E2 7135.331} C_VEL
LIN {X 0,Y 473.902,Z 326.725,A -85,B 0,C 180,E1 7135.925,E2 7135.925} C_VEL
LIN {X 0,Y 464.857,Z 297.81,A -85,B 0,C 180,E1 7136.889,E2 7136.889} C_VEL
LIN {X 0,Y 464.629,Z 297.81,A -85,B 0,C 180,E1 7143.512,E2 7143.512} C_VEL
LIN {X 0,Y 464.417,Z 297.81,A -85,B 0,C 180,E1 7150.529,E2 7150.529} C_VEL
LIN {X 0,Y 464.54,Z 297.81,A -85,B 0,C 180,E1 7157.002,E2 7157.002} C_VEL
LIN {X 0,Y 464.587,Z 297.81,A -85,B 0,C 180,E1 7161.907,E2 7161.907} C_VEL
LIN {X 0,Y 464.583,Z 297.81,A -85,B 0,C 180,E1 7168.701,E2 7168.701} C_VEL
LIN {X 0,Y 464.841,Z 297.81,A -85,B 0,C 180,E1 7175.36,E2 7175.36} C_VEL
LIN {X 0,Y 464.98,Z 297.81,A -85,B 0,C 180,E1 7181.075,E2 7181.075} C_VEL
LIN {X 0,Y 464.935,Z 297.81,A -85,B 0,C 180,E1 7186.88,E2 7186.88} C_VEL
LIN {X 0,Y 465.271,Z 297.81,A -85,B 0,C 180,E1 7192.557,E2 7192.557} C_VEL
LIN {X 0,Y 465.601,Z 297.81,A -85,B 0,C 180,E1 7198.154,E2 7198.154} C_VEL
LIN {X 0,Y 465.437,Z 297.81,A -85,B 0,C 180,E1 7203.73,E2 7203.73} C_VEL
LIN {X 0,Y 465.23,Z 297.81,A -85,B 0,C 180,E1 7209.345,E2 7209.345} C_VEL
LIN {X 0,Y 465.088,Z 297.81,A -85,B 0,C 180,E1 7215.057,E2 7215.057} C_VEL
LIN {X 0,Y 464.946,Z 297.81,A -85,B 0,C 180,E1 7220.93,E2 7220.93} C_VEL
LIN {X 0,Y 464.752,Z 297.81,A -85,B 0,C 180,E1 7227.051,E2 7227.051} C_VEL
LIN {X 0,Y 464.973,Z 298.234,A -85,B 0,C 180,E1 7233.064,E2 7233.064} C_VEL
LIN {X 0,Y 471.701,Z 325.183,A -85,B 0,C 180,E1 7234.51,E2 7234.51} C_VEL
LIN {X 0,Y 470.437,Z 350.536,A -85,B 0,C 180,E1 7236.291,E2 7236.291} C_VEL
LIN {X 0,Y 469.092,Z 371.089,A -85,B 0,C 180,E1 7238.533,E2 7238.533} C_VEL
LIN {X 0,Y 467.898,Z 387.94,A -85,B 0,C 180,E1 7241.311,E2 7241.311} C_VEL
LIN {X 0,Y 467.265,Z 398.544,A -85,B 0,C 180,E1 7244.06,E2 7244.06} C_VEL
LIN {X 0,Y 466.716,Z 405.22,A -85,B 0,C 180,E1 7247.237,E2 7247.237} C_VEL
LIN {X 0,Y 466.46,Z 406.527,A -85,B 0,C 180,E1 7250.953,E2 7250.953} C_VEL
LIN {X 0,Y 466.815,Z 401.568,A -85,B 0,C 180,E1 7254.419,E2 7254.419} C_VEL
LIN {X 0,Y 467.522,Z 390.542,A -85,B 0,C 180,E1 7257.74,E2 7257.74} C_VEL
LIN {X 0,Y 468.438,Z 374.896,A -85,B 0,C 180,E1 7260.573,E2 7260.573} C_VEL
LIN {X 0,Y 469.641,Z 354.94,A -85,B 0,C 180,E1 7262.954,E2 7262.954} C_VEL
LIN {X 0,Y 470.798,Z 330.227,A -85,B 0,C 180,E1 7264.867,E2 7264.867} C_VEL
LIN {X 0,Y 470.082,Z 317.667,A -85,B 0,C 180,E1 7265.589,E2 7265.589} C_VEL
LIN {X 0,Y 465.062,Z 297.81,A -85,B 0,C 180,E1 7266.58,E2 7266.58} C_VEL
LIN {X 0,Y 465.057,Z 297.81,A -85,B 0,C 180,E1 7273.021,E2 7273.021} C_VEL
LIN {X 0,Y 465.234,Z 298.084,A -85,B 0,C 180,E1 7279.996,E2 7279.996} C_VEL
LIN {X 0,Y 470.205,Z 324.467,A -85,B 0,C 180,E1 7281.061,E2 7281.061} C_VEL
LIN {X 0,Y 469.511,Z 348.71,A -85,B 0,C 180,E1 7282.614,E2 7282.614} C_VEL
LIN {X 0,Y 468.568,Z 369.148,A -85,B 0,C 180,E1 7284.688,E2 7284.688} C_VEL
LIN {X 0,Y 467.725,Z 385.673,A -85,B 0,C 180,E1 7287.227,E2 7287.227} C_VEL
LIN {X 0,Y 467.094,Z 397.25,A -85,B 0,C 180,E1 7290.001,E2 7290.001} C_VEL
LIN {X 0,Y 466.814,Z 403.948,A -85,B 0,C 180,E1 7292.78,E2 7292.78} C_VEL
LIN {X 0,Y 466.568,Z 406.574,A -85,B 0,C 180,E1 7295.569,E2 7295.569} C_VEL
LIN {X 0,Y 466.654,Z 405.283,A -85,B 0,C 180,E1 7298.368,E2 7298.368} C_VEL
LIN {X 0,Y 467.162,Z 398.609,A -85,B 0,C 180,E1 7301.648,E2 7301.648} C_VEL
LIN {X 0,Y 467.825,Z 386.325,A -85,B 0,C 180,E1 7304.738,E2 7304.738} C_VEL
LIN {X 0,Y 468.831,Z 369.016,A -85,B 0,C 180,E1 7307.425,E2 7307.425} C_VEL
LIN {X 0,Y 469.967,Z 347.439,A -85,B 0,C 180,E1 7309.581,E2 7309.581} C_VEL
LIN {X 0,Y 470.691,Z 322.543,A -85,B 0,C 180,E1 7311.119,E2 7311.119} C_VEL
LIN {X 0,Y 465.027,Z 297.81,A -85,B 0,C 180,E1 7312.204,E2 7312.204} C_VEL
LIN {X 0,Y 464.644,Z 297.81,A -85,B 0,C 180,E1 7319.154,E2 7319.154} C_VEL
LIN {X 0,Y 464.68,Z 297.81,A -85,B 0,C 180,E1 7325.77,E2 7325.77} C_VEL
LIN {X 0,Y 464.521,Z 297.81,A -85,B 0,C 180,E1 7331.636,E2 7331.636} C_VEL
LIN {X 0,Y 464.565,Z 297.81,A -85,B 0,C 180,E1 7338.339,E2 7338.339} C_VEL
LIN {X 0,Y 464.641,Z 297.81,A -85,B 0,C 180,E1 7344.284,E2 7344.284} C_VEL
LIN {X 0,Y 464.68,Z 297.81,A -85,B 0,C 180,E1 7351.259,E2 7351.259} C_VEL
LIN {X 0,Y 464.865,Z 297.81,A -85,B 0,C 180,E1 7357.061,E2 7357.061} C_VEL
LIN {X 0,Y 465.053,Z 297.81,A -85,B 0,C 180,E1 7363.008,E2 7363.008} C_VEL
LIN {X 0,Y 465.07,Z 297.81,A -85,B 0,C 180,E1 7368.762,E2 7368.762} C_VEL
LIN {X 0,Y 465.375,Z 297.81,A -85,B 0,C 180,E1 7374.406,E2 7374.406} C_VEL
LIN {X 0,Y 465.572,Z 297.81,A -85,B 0,C 180,E1 7379.988,E2 7379.988} C_VEL
LIN {X 0,Y 465.357,Z 297.81,A -85,B 0,C 180,E1 7385.571,E2 7385.571} C_VEL
LIN {X 0,Y 465.183,Z 297.81,A -85,B 0,C 180,E1 7391.212,E2 7391.212} C_VEL
LIN {X 0,Y 465.04,Z 297.81,A -85,B 0,C 180,E1 7396.968,E2 7396.968} C_VEL
LIN {X 0,Y 464.893,Z 297.81,A -85,B 0,C 180,E1 7402.912,E2 7402.912} C_VEL
LIN {X 0,Y 464.708,Z 297.81,A -85,B 0,C 180,E1 7409.136,E2 7409.136} C_VEL
LIN {X 0,Y 464.605,Z 297.81,A -85,B 0,C 180,E1 7415.763,E2 7415.763} C_VEL
LIN {X 0,Y 464.489,Z 297.81,A -85,B 0,C 180,E1 7421.65,E2 7421.65} C_VEL
LIN {X 0,Y 464.595,Z 297.81,A -85,B 0,C 180,E1 7428.319,E2 7428.319} C_VEL
LIN {X 0,Y 464.673,Z 297.81,A -85,B 0,C 180,E1 7434.261,E2 7434.261} C_VEL
LIN {X 0,Y 464.811,Z 297.81,A -85,B 0,C 180,E1 7441.208,E2 7441.208} C_VEL
LIN {X 0,Y 464.826,Z 297.81,A -85,B 0,C 180,E1 7442.14,E2 7442.14} C_VEL
LIN {X 0,Y 464.993,Z 301.123,A -85,B 0,C 180,E1 7442.864,E2 7442.864} C_VEL
LIN {X 0,Y 465.35,Z 311.096,A -85,B 0,C 180,E1 7443.388,E2 7443.388} C_VEL
LIN {X 0,Y 467.167,Z 330.047,A -85,B 0,C 180,E1 7443.77,E2 7443.77} C_VEL
LIN {X 0,Y 466.812,Z 374.575,A -85,B 0,C 180,E1 7444.632,E2 7444.632} C_VEL
LIN {X 0,Y 465.038,Z 408.13,A -85,B 0,C 180,E1 7446.006,E2 7446.006} C_VEL
LIN {X 0,Y 462.986,Z 438.777,A -85,B 0,C 180,E1 7448.032,E2 7448.032} C_VEL
LIN {X 0,Y 460.932,Z 467.094,A -85,B 0,C 180,E1 7450.766,E2 7450.766} C_VEL
LIN {X 0,Y 459.406,Z 491.222,A -85,B 0,C 180,E1 7454.032,E2 7454.032} C_VEL
LIN {X 0,Y 458.509,Z 510.342,A -85,B 0,C 180,E1 7457.647,E2 7457.647} C_VEL
LIN {X 0,Y 458.271,Z 524.836,A -85,B 0,C 180,E1 7461.71,E2 7461.71} C_VEL
LIN {X 0,Y 458.308,Z 532.558,A -85,B 0,C 180,E1 7465.278,E2 7465.278} C_VEL
LIN {X 0,Y 458.42,Z 535.555,A -85,B 0,C 180,E1 7468.113,E2 7468.113} C_VEL
LIN {X 0,Y 458.396,Z 535.476,A -85,B 0,C 180,E1 7471.886,E2 7471.886} C_VEL
LIN {X 0,Y 458.36,Z 530.71,A -85,B 0,C 180,E1 7475.668,E2 7475.668} C_VEL
LIN {X 0,Y 458.332,Z 520.886,A -85,B 0,C 180,E1 7479.475,E2 7479.475} C_VEL
LIN {X 0,Y 458.683,Z 505.323,A -85,B 0,C 180,E1 7483.314,E2 7483.314} C_VEL
LIN {X 0,Y 459.761,Z 484.14,A -85,B 0,C 180,E1 7486.935,E2 7486.935} C_VEL
LIN {X 0,Y 461.477,Z 458.434,A -85,B 0,C 180,E1 7490.08,E2 7490.08} C_VEL
LIN {X 0,Y 463.478,Z 429.684,A -85,B 0,C 180,E1 7492.586,E2 7492.586} C_VEL
LIN {X 0,Y 465.554,Z 397.404,A -85,B 0,C 180,E1 7494.473,E2 7494.473} C_VEL
LIN {X 0,Y 466.97,Z 364.969,A -85,B 0,C 180,E1 7495.595,E2 7495.595} C_VEL
LIN {X 0,Y 466.856,Z 329.172,A -85,B 0,C 180,E1 7496.233,E2 7496.233} C_VEL
LIN {X 0,Y 456.897,Z 297.81,A -85,B 0,C 180,E1 7497.299,E2 7497.299} C_VEL
LIN {X 0,Y 456.633,Z 297.81,A -85,B 0,C 180,E1 7504.313,E2 7504.313} C_VEL
LIN {X 0,Y 456.531,Z 297.81,A -85,B 0,C 180,E1 7510.531,E2 7510.531} C_VEL
LIN {X 0,Y 456.63,Z 297.81,A -85,B 0,C 180,E1 7516.636,E2 7516.636} C_VEL
LIN {X 0,Y 456.646,Z 297.81,A -85,B 0,C 180,E1 7522.474,E2 7522.474} C_VEL
LIN {X 0,Y 456.647,Z 297.81,A -85,B 0,C 180,E1 7529.223,E2 7529.223} C_VEL
LIN {X 0,Y 456.833,Z 297.81,A -85,B 0,C 180,E1 7534.582,E2 7534.582} C_VEL
LIN {X 0,Y 457.051,Z 297.81,A -85,B 0,C 180,E1 7540.733,E2 7540.733} C_VEL
LIN {X 0,Y 457.039,Z 297.81,A -85,B 0,C 180,E1 7546.649,E2 7546.649} C_VEL
LIN {X 0,Y 457.343,Z 297.81,A -85,B 0,C 180,E1 7552.428,E2 7552.428} C_VEL
LIN {X 0,Y 457.691,Z 297.81,A -85,B 0,C 180,E1 7558.122,E2 7558.122} C_VEL
LIN {X 0,Y 457.524,Z 297.81,A -85,B 0,C 180,E1 7563.794,E2 7563.794} C_VEL
LIN {X 0,Y 457.311,Z 297.81,A -85,B 0,C 180,E1 7569.509,E2 7569.509} C_VEL
LIN {X 0,Y 457.151,Z 297.81,A -85,B 0,C 180,E1 7575.324,E2 7575.324} C_VEL
LIN {X 0,Y 456.988,Z 297.81,A -85,B 0,C 180,E1 7581.312,E2 7581.312} C_VEL
LIN {X 0,Y 456.83,Z 297.81,A -85,B 0,C 180,E1 7587.559,E2 7587.559} C_VEL
LIN {X 0,Y 457.003,Z 297.81,A -85,B 0,C 180,E1 7592.626,E2 7592.626} C_VEL
LIN {X 0,Y 464.164,Z 325.214,A -85,B 0,C 180,E1 7594.137,E2 7594.137} C_VEL
LIN {X 0,Y 462.988,Z 350.656,A -85,B 0,C 180,E1 7595.936,E2 7595.936} C_VEL
LIN {X 0,Y 461.493,Z 372.165,A -85,B 0,C 180,E1 7598.303,E2 7598.303} C_VEL
LIN {X 0,Y 460.261,Z 388.64,A -85,B 0,C 180,E1 7601.057,E2 7601.057} C_VEL
LIN {X 0,Y 459.577,Z 399.065,A -85,B 0,C 180,E1 7603.751,E2 7603.751} C_VEL
LIN {X 0,Y 458.905,Z 406.361,A -85,B 0,C 180,E1 7607.201,E2 7607.201} C_VEL
LIN {X 0,Y 458.704,Z 407.887,A -85,B 0,C 180,E1 7609.188,E2 7609.188} C_VEL
LIN {X 0,Y 458.735,Z 406.619,A -85,B 0,C 180,E1 7612.158,E2 7612.158} C_VEL
LIN {X 0,Y 459.275,Z 399.549,A -85,B 0,C 180,E1 7615.656,E2 7615.656} C_VEL
LIN {X 0,Y 460.071,Z 386.806,A -85,B 0,C 180,E1 7618.893,E2 7618.893} C_VEL
LIN {X 0,Y 461.236,Z 368.615,A -85,B 0,C 180,E1 7621.763,E2 7621.763} C_VEL
LIN {X 0,Y 462.644,Z 345.364,A -85,B 0,C 180,E1 7624.129,E2 7624.129} C_VEL
LIN {X 0,Y 463.038,Z 321.466,A -85,B 0,C 180,E1 7625.706,E2 7625.706} C_VEL
LIN {X 0,Y 457.138,Z 297.81,A -85,B 0,C 180,E1 7626.954,E2 7626.954} C_VEL
LIN {X 0,Y 457.133,Z 297.81,A -85,B 0,C 180,E1 7633.241,E2 7633.241} C_VEL
LIN {X 0,Y 457.308,Z 297.81,A -85,B 0,C 180,E1 7639.712,E2 7639.712} C_VEL
LIN {X 0,Y 462.611,Z 324.345,A -85,B 0,C 180,E1 7640.782,E2 7640.782} C_VEL
LIN {X 0,Y 461.865,Z 349.27,A -85,B 0,C 180,E1 7642.373,E2 7642.373} C_VEL
LIN {X 0,Y 460.833,Z 370.807,A -85,B 0,C 180,E1 7644.599,E2 7644.599} C_VEL
LIN {X 0,Y 459.944,Z 387.144,A -85,B 0,C 180,E1 7647.18,E2 7647.18} C_VEL
LIN {X 0,Y 459.28,Z 398.567,A -85,B 0,C 180,E1 7650.001,E2 7650.001} C_VEL
LIN {X 0,Y 458.977,Z 405.152,A -85,B 0,C 180,E1 7652.827,E2 7652.827} C_VEL
LIN {X 0,Y 458.734,Z 407.67,A -85,B 0,C 180,E1 7655.664,E2 7655.664} C_VEL
LIN {X 0,Y 458.868,Z 406.292,A -85,B 0,C 180,E1 7658.49,E2 7658.49} C_VEL
LIN {X 0,Y 459.417,Z 399.449,A -85,B 0,C 180,E1 7661.847,E2 7661.847} C_VEL
LIN {X 0,Y 460.17,Z 387.001,A -85,B 0,C 180,E1 7664.989,E2 7664.989} C_VEL
LIN {X 0,Y 461.209,Z 369.981,A -85,B 0,C 180,E1 7667.657,E2 7667.657} C_VEL
LIN {X 0,Y 462.388,Z 349.03,A -85,B 0,C 180,E1 7669.791,E2 7669.791} C_VEL
LIN {X 0,Y 463.23,Z 324.139,A -85,B 0,C 180,E1 7671.37,E2 7671.37} C_VEL
LIN {X 0,Y 457.055,Z 297.81,A -85,B 0,C 180,E1 7672.564,E2 7672.564} C_VEL
LIN {X 0,Y 456.787,Z 297.81,A -85,B 0,C 180,E1 7677.548,E2 7677.548} C_VEL
LIN {X 0,Y 456.661,Z 297.81,A -85,B 0,C 180,E1 7684.276,E2 7684.276} C_VEL
LIN {X 0,Y 456.664,Z 297.81,A -85,B 0,C 180,E1 7690.515,E2 7690.515} C_VEL
LIN {X 0,Y 456.652,Z 297.81,A -85,B 0,C 180,E1 7696.635,E2 7696.635} C_VEL
LIN {X 0,Y 456.645,Z 297.81,A -85,B 0,C 180,E1 7702.476,E2 7702.476} C_VEL
LIN {X 0,Y 456.619,Z 297.81,A -85,B 0,C 180,E1 7709.231,E2 7709.231} C_VEL
LIN {X 0,Y 456.801,Z 297.81,A -85,B 0,C 180,E1 7714.554,E2 7714.554} C_VEL
LIN {X 0,Y 457.114,Z 297.81,A -85,B 0,C 180,E1 7720.711,E2 7720.711} C_VEL
LIN {X 0,Y 457.097,Z 297.81,A -85,B 0,C 180,E1 7726.626,E2 7726.626} C_VEL
LIN {X 0,Y 457.362,Z 297.81,A -85,B 0,C 180,E1 7732.978,E2 7732.978} C_VEL
LIN {X 0,Y 457.703,Z 297.81,A -85,B 0,C 180,E1 7738.099,E2 7738.099} C_VEL
LIN {X 0,Y 457.573,Z 297.81,A -85,B 0,C 180,E1 7743.77,E2 7743.77} C_VEL
LIN {X 0,Y 457.366,Z 297.81,A -85,B 0,C 180,E1 7749.484,E2 7749.484} C_VEL
LIN {X 0,Y 457.146,Z 297.81,A -85,B 0,C 180,E1 7755.3,E2 7755.3} C_VEL
LIN {X 0,Y 457.006,Z 297.81,A -85,B 0,C 180,E1 7761.286,E2 7761.286} C_VEL
LIN {X 0,Y 456.814,Z 297.81,A -85,B 0,C 180,E1 7767.534,E2 7767.534} C_VEL
LIN {X 0,Y 456.635,Z 297.81,A -85,B 0,C 180,E1 7774.294,E2 7774.294} C_VEL
LIN {X 0,Y 456.586,Z 297.81,A -85,B 0,C 180,E1 7780.523,E2 7780.523} C_VEL
LIN {X 0,Y 456.682,Z 297.81,A -85,B 0,C 180,E1 7786.615,E2 7786.615} C_VEL
LIN {X 0,Y 456.685,Z 297.81,A -85,B 0,C 180,E1 7792.451,E2 7792.451} C_VEL
LIN {X 0,Y 456.725,Z 297.81,A -85,B 0,C 180,E1 7799.188,E2 7799.188} C_VEL
LIN {X 0,Y 457.047,Z 298.354,A -85,B 0,C 180,E1 7802.78,E2 7802.78} C_VEL
LIN {X 0,Y 467.167,Z 330.047,A -85,B 0,C 180,E1 7803.77,E2 7803.77} C_VEL
LIN {X 0,Y 466.796,Z 340.685,A -85,B 0,C 180,E1 7803.912,E2 7803.912} C_VEL
LIN {X 0,Y 459.808,Z 362.096,A -85,B 0,C 180,E1 7803.969,E2 7803.969} C_VEL
LIN {X 0,Y 459.654,Z 364.314,A -85,B 0,C 180,E1 7804.019,E2 7804.019} C_VEL
LIN {X 0,Y 458.018,Z 398.717,A -85,B 0,C 180,E1 7805.226,E2 7805.226} C_VEL
LIN {X 0,Y 455.859,Z 430.704,A -85,B 0,C 180,E1 7807.153,E2 7807.153} C_VEL
LIN {X 0,Y 453.706,Z 460.208,A -85,B 0,C 180,E1 7809.814,E2 7809.814} C_VEL
LIN {X 0,Y 451.934,Z 485.229,A -85,B 0,C 180,E1 7813.012,E2 7813.012} C_VEL
LIN {X 0,Y 450.808,Z 505.818,A -85,B 0,C 180,E1 7816.695,E2 7816.695} C_VEL
LIN {X 0,Y 450.395,Z 520.108,A -85,B 0,C 180,E1 7820.356,E2 7820.356} C_VEL
LIN {X 0,Y 450.473,Z 529.828,A -85,B 0,C 180,E1 7824.232,E2 7824.232} C_VEL
LIN {X 0,Y 450.588,Z 534.462,A -85,B 0,C 180,E1 7828.08,E2 7828.08} C_VEL
LIN {X 0,Y 450.568,Z 534.377,A -85,B 0,C 180,E1 7831.919,E2 7831.919} C_VEL
LIN {X 0,Y 450.5,Z 529.588,A -85,B 0,C 180,E1 7835.767,E2 7835.767} C_VEL
LIN {X 0,Y 450.442,Z 519.718,A -85,B 0,C 180,E1 7839.642,E2 7839.642} C_VEL
LIN {X 0,Y 450.862,Z 504.114,A -85,B 0,C 180,E1 7843.549,E2 7843.549} C_VEL
LIN {X 0,Y 451.974,Z 482.845,A -85,B 0,C 180,E1 7847.235,E2 7847.235} C_VEL
LIN {X 0,Y 453.848,Z 457.017,A -85,B 0,C 180,E1 7850.433,E2 7850.433} C_VEL
LIN {X 0,Y 456.004,Z 427.612,A -85,B 0,C 180,E1 7853.012,E2 7853.012} C_VEL
LIN {X 0,Y 458.22,Z 395.14,A -85,B 0,C 180,E1 7854.906,E2 7854.906} C_VEL
LIN {X 0,Y 459.698,Z 362.381,A -85,B 0,C 180,E1 7856.013,E2 7856.013} C_VEL
LIN {X 0,Y 459.287,Z 329.927,A -85,B 0,C 180,E1 7856.607,E2 7856.607} C_VEL
LIN {X 0,Y 448.944,Z 297.81,A -85,B 0,C 180,E1 7857.767,E2 7857.767} C_VEL
LIN {X 0,Y 448.664,Z 297.81,A -85,B 0,C 180,E1 7864.873,E2 7864.873} C_VEL
LIN {X 0,Y 448.616,Z 297.81,A -85,B 0,C 180,E1 7869.724,E2 7869.724} C_VEL
LIN {X 0,Y 448.602,Z 297.81,A -85,B 0,C 180,E1 7875.073,E2 7875.073} C_VEL
LIN {X 0,Y 448.729,Z 297.81,A -85,B 0,C 180,E1 7880.664,E2 7880.664} C_VEL
LIN {X 0,Y 448.67,Z 297.81,A -85,B 0,C 180,E1 7887.457,E2 7887.457} C_VEL
LIN {X 0,Y 448.918,Z 297.81,A -85,B 0,C 180,E1 7894.101,E2 7894.101} C_VEL
LIN {X 0,Y 449.096,Z 297.81,A -85,B 0,C 180,E1 7900.378,E2 7900.378} C_VEL
LIN {X 0,Y 449.132,Z 297.81,A -85,B 0,C 180,E1 7906.991,E2 7906.991} C_VEL
LIN {X 0,Y 449.429,Z 297.81,A -85,B 0,C 180,E1 7912.294,E2 7912.294} C_VEL
LIN {X 0,Y 449.806,Z 297.81,A -85,B 0,C 180,E1 7918.089,E2 7918.089} C_VEL
LIN {X 0,Y 449.61,Z 297.81,A -85,B 0,C 180,E1 7923.861,E2 7923.861} C_VEL
LIN {X 0,Y 449.381,Z 297.81,A -85,B 0,C 180,E1 7929.678,E2 7929.678} C_VEL
LIN {X 0,Y 449.254,Z 297.81,A -85,B 0,C 180,E1 7935.601,E2 7935.601} C_VEL
LIN {X 0,Y 449.059,Z 297.81,A -85,B 0,C 180,E1 7941.707,E2 7941.707} C_VEL
LIN {X 0,Y 448.858,Z 297.81,A -85,B 0,C 180,E1 7948.092,E2 7948.092} C_VEL
LIN {X 0,Y 449.037,Z 297.81,A -85,B 0,C 180,E1 7952.184,E2 7952.184} C_VEL
LIN {X 0,Y 456.66,Z 326.452,A -85,B 0,C 180,E1 7953.822,E2 7953.822} C_VEL
LIN {X 0,Y 455.501,Z 351.691,A -85,B 0,C 180,E1 7955.651,E2 7955.651} C_VEL
LIN {X 0,Y 453.891,Z 373.346,A -85,B 0,C 180,E1 7958.079,E2 7958.079} C_VEL
LIN {X 0,Y 452.575,Z 389.778,A -85,B 0,C 180,E1 7960.879,E2 7960.879} C_VEL
LIN {X 0,Y 451.675,Z 401.817,A -85,B 0,C 180,E1 7964.2,E2 7964.2} C_VEL
LIN {X 0,Y 451.056,Z 407.794,A -85,B 0,C 180,E1 7967.412,E2 7967.412} C_VEL
LIN {X 0,Y 450.849,Z 408.457,A -85,B 0,C 180,E1 7971.375,E2 7971.375} C_VEL
LIN {X 0,Y 451.336,Z 402.723,A -85,B 0,C 180,E1 7974.965,E2 7974.965} C_VEL
LIN {X 0,Y 452.115,Z 391.412,A -85,B 0,C 180,E1 7978.29,E2 7978.29} C_VEL
LIN {X 0,Y 453.322,Z 374.405,A -85,B 0,C 180,E1 7981.318,E2 7981.318} C_VEL
LIN {X 0,Y 454.675,Z 352.629,A -85,B 0,C 180,E1 7983.829,E2 7983.829} C_VEL
LIN {X 0,Y 455.987,Z 327.326,A -85,B 0,C 180,E1 7985.696,E2 7985.696} C_VEL
LIN {X 0,Y 449.728,Z 300.56,A -85,B 0,C 180,E1 7987.168,E2 7987.168} C_VEL
LIN {X 0,Y 449.21,Z 297.81,A -85,B 0,C 180,E1 7987.34,E2 7987.34} C_VEL
LIN {X 0,Y 449.187,Z 297.81,A -85,B 0,C 180,E1 7992.402,E2 7992.402} C_VEL
LIN {X 0,Y 449.344,Z 297.81,A -85,B 0,C 180,E1 7999.432,E2 7999.432} C_VEL
LIN {X 0,Y 454.988,Z 324.465,A -85,B 0,C 180,E1 8000.506,E2 8000.506} C_VEL
LIN {X 0,Y 454.296,Z 348.594,A -85,B 0,C 180,E1 8002.024,E2 8002.024} C_VEL
LIN {X 0,Y 453.22,Z 370.634,A -85,B 0,C 180,E1 8004.268,E2 8004.268} C_VEL
LIN {X 0,Y 452.263,Z 387.371,A -85,B 0,C 180,E1 8006.893,E2 8006.893} C_VEL
LIN {X 0,Y 451.475,Z 399.877,A -85,B 0,C 180,E1 8010.001,E2 8010.001} C_VEL
LIN {X 0,Y 451.169,Z 406.349,A -85,B 0,C 180,E1 8012.876,E2 8012.876} C_VEL
LIN {X 0,Y 450.907,Z 408.766,A -85,B 0,C 180,E1 8015.763,E2 8015.763} C_VEL
LIN {X 0,Y 451.048,Z 407.474,A -85,B 0,C 180,E1 8018.475,E2 8018.475} C_VEL
LIN {X 0,Y 451.654,Z 400.297,A -85,B 0,C 180,E1 8022.053,E2 8022.053} C_VEL
LIN {X 0,Y 452.484,Z 388.017,A -85,B 0,C 180,E1 8025.183,E2 8025.183} C_VEL
LIN {X 0,Y 453.646,Z 370.011,A -85,B 0,C 180,E1 8028.019,E2 8028.019} C_VEL
LIN {X 0,Y 455.017,Z 347.658,A -85,B 0,C 180,E1 8030.252,E2 8030.252} C_VEL
LIN {X 0,Y 455.244,Z 322.294,A -85,B 0,C 180,E1 8031.821,E2 8031.821} C_VEL
LIN {X 0,Y 449.106,Z 297.81,A -85,B 0,C 180,E1 8032.891,E2 8032.891} C_VEL
LIN {X 0,Y 448.733,Z 297.81,A -85,B 0,C 180,E1 8039.006,E2 8039.006} C_VEL
LIN {X 0,Y 448.716,Z 297.81,A -85,B 0,C 180,E1 8044.869,E2 8044.869} C_VEL
LIN {X 0,Y 448.756,Z 297.81,A -85,B 0,C 180,E1 8049.71,E2 8049.71} C_VEL
LIN {X 0,Y 448.643,Z 297.81,A -85,B 0,C 180,E1 8055.044,E2 8055.044} C_VEL
LIN {X 0,Y 448.758,Z 297.81,A -85,B 0,C 180,E1 8060.661,E2 8060.661} C_VEL
LIN {X 0,Y 448.658,Z 297.81,A -85,B 0,C 180,E1 8067.428,E2 8067.428} C_VEL
LIN {X 0,Y 448.889,Z 297.81,A -85,B 0,C 180,E1 8074.072,E2 8074.072} C_VEL
LIN {X 0,Y 449.157,Z 297.81,A -85,B 0,C 180,E1 8080.356,E2 8080.356} C_VEL
LIN {X 0,Y 449.197,Z 297.81,A -85,B 0,C 180,E1 8086.96,E2 8086.96} C_VEL
LIN {X 0,Y 449.454,Z 297.81,A -85,B 0,C 180,E1 8092.979,E2 8092.979} C_VEL
LIN {X 0,Y 449.819,Z 297.81,A -85,B 0,C 180,E1 8098.065,E2 8098.065} C_VEL
LIN {X 0,Y 449.659,Z 297.81,A -85,B 0,C 180,E1 8103.837,E2 8103.837} C_VEL
LIN {X 0,Y 449.436,Z 297.81,A -85,B 0,C 180,E1 8109.653,E2 8109.653} C_VEL
LIN {X 0,Y 449.25,Z 297.81,A -85,B 0,C 180,E1 8115.576,E2 8115.576} C_VEL
LIN {X 0,Y 449.081,Z 297.81,A -85,B 0,C 180,E1 8121.68,E2 8121.68} C_VEL
LIN {X 0,Y 448.832,Z 297.81,A -85,B 0,C 180,E1 8128.066,E2 8128.066} C_VEL
LIN {X 0,Y 448.673,Z 297.81,A -85,B 0,C 180,E1 8134.859,E2 8134.859} C_VEL
LIN {X 0,Y 448.661,Z 297.81,A -85,B 0,C 180,E1 8139.706,E2 8139.706} C_VEL
LIN {X 0,Y 448.667,Z 297.81,A -85,B 0,C 180,E1 8145.065,E2 8145.065} C_VEL
LIN {X 0,Y 448.812,Z 297.81,A -85,B 0,C 180,E1 8150.635,E2 8150.635} C_VEL
LIN {X 0,Y 448.74,Z 297.81,A -85,B 0,C 180,E1 8157.449,E2 8157.449} C_VEL
LIN {X 0,Y 449.103,Z 298.399,A -85,B 0,C 180,E1 8162.377,E2 8162.377} C_VEL
LIN {X 0,Y 459.983,Z 332.191,A -85,B 0,C 180,E1 8163.459,E2 8163.459} C_VEL
LIN {X 0,Y 459.654,Z 364.314,A -85,B 0,C 180,E1 8164.019,E2 8164.019} C_VEL
LIN {X 0,Y 455.376,Z 381.14,A -85,B 0,C 180,E1 8164.34,E2 8164.34} C_VEL
LIN {X 0,Y 450.608,Z 397.529,A -85,B 0,C 180,E1 8164.853,E2 8164.853} C_VEL
LIN {X 0,Y 448.286,Z 429.999,A -85,B 0,C 180,E1 8166.832,E2 8166.832} C_VEL
LIN {X 0,Y 446.082,Z 458.695,A -85,B 0,C 180,E1 8169.453,E2 8169.453} C_VEL
LIN {X 0,Y 444.185,Z 483.902,A -85,B 0,C 180,E1 8172.706,E2 8172.706} C_VEL
LIN {X 0,Y 442.998,Z 504.612,A -85,B 0,C 180,E1 8176.456,E2 8176.456} C_VEL
LIN {X 0,Y 442.519,Z 520.09,A -85,B 0,C 180,E1 8180.541,E2 8180.541} C_VEL
LIN {X 0,Y 442.621,Z 528.719,A -85,B 0,C 180,E1 8184.129,E2 8184.129} C_VEL
LIN {X 0,Y 442.761,Z 533.371,A -85,B 0,C 180,E1 8188.046,E2 8188.046} C_VEL
LIN {X 0,Y 442.742,Z 533.283,A -85,B 0,C 180,E1 8191.953,E2 8191.953} C_VEL
LIN {X 0,Y 442.646,Z 528.47,A -85,B 0,C 180,E1 8195.869,E2 8195.869} C_VEL
LIN {X 0,Y 442.573,Z 518.558,A -85,B 0,C 180,E1 8199.815,E2 8199.815} C_VEL
LIN {X 0,Y 443.026,Z 502.91,A -85,B 0,C 180,E1 8203.793,E2 8203.793} C_VEL
LIN {X 0,Y 444.225,Z 481.563,A -85,B 0,C 180,E1 8207.546,E2 8207.546} C_VEL
LIN {X 0,Y 446.197,Z 455.614,A -85,B 0,C 180,E1 8210.799,E2 8210.799} C_VEL
LIN {X 0,Y 448.536,Z 426.029,A -85,B 0,C 180,E1 8213.415,E2 8213.415} C_VEL
LIN {X 0,Y 450.86,Z 393.933,A -85,B 0,C 180,E1 8215.303,E2 8215.303} C_VEL
LIN {X 0,Y 452.435,Z 361.074,A -85,B 0,C 180,E1 8216.414,E2 8216.414} C_VEL
LIN {X 0,Y 452.072,Z 331.665,A -85,B 0,C 180,E1 8216.962,E2 8216.962} C_VEL
LIN {X 0,Y 440.978,Z 297.81,A -85,B 0,C 180,E1 8218.259,E2 8218.259} C_VEL
LIN {X 0,Y 440.733,Z 297.81,A -85,B 0,C 180,E1 8225.594,E2 8225.594} C_VEL
LIN {X 0,Y 440.593,Z 297.81,A -85,B 0,C 180,E1 8231.124,E2 8231.124} C_VEL
LIN {X 0,Y 440.663,Z 297.81,A -85,B 0,C 180,E1 8236.789,E2 8236.789} C_VEL
LIN {X 0,Y 440.765,Z 297.81,A -85,B 0,C 180,E1 8241.972,E2 8241.972} C_VEL
LIN {X 0,Y 440.722,Z 297.81,A -85,B 0,C 180,E1 8246.795,E2 8246.795} C_VEL
LIN {X 0,Y 440.935,Z 297.81,A -85,B 0,C 180,E1 8253.596,E2 8253.596} C_VEL
LIN {X 0,Y 441.164,Z 297.81,A -85,B 0,C 180,E1 8260.011,E2 8260.011} C_VEL
LIN {X 0,Y 441.166,Z 297.81,A -85,B 0,C 180,E1 8266.159,E2 8266.159} C_VEL
LIN {X 0,Y 441.55,Z 297.81,A -85,B 0,C 180,E1 8272.335,E2 8272.335} C_VEL
LIN {X 0,Y 441.895,Z 297.81,A -85,B 0,C 180,E1 8278.055,E2 8278.055} C_VEL
LIN {X 0,Y 441.697,Z 297.81,A -85,B 0,C 180,E1 8283.93,E2 8283.93} C_VEL
LIN {X 0,Y 441.478,Z 297.81,A -85,B 0,C 180,E1 8289.853,E2 8289.853} C_VEL
LIN {X 0,Y 441.305,Z 297.81,A -85,B 0,C 180,E1 8295.889,E2 8295.889} C_VEL
LIN {X 0,Y 441.051,Z 297.81,A -85,B 0,C 180,E1 8302.518,E2 8302.518} C_VEL
LIN {X 0,Y 440.953,Z 297.81,A -85,B 0,C 180,E1 8308.641,E2 8308.641} C_VEL
LIN {X 0,Y 441.073,Z 297.81,A -85,B 0,C 180,E1 8311.721,E2 8311.721} C_VEL
LIN {X 0,Y 449.027,Z 327.021,A -85,B 0,C 180,E1 8313.442,E2 8313.442} C_VEL
LIN {X 0,Y 448.083,Z 352.344,A -85,B 0,C 180,E1 8315.318,E2 8315.318} C_VEL
LIN {X 0,Y 446.377,Z 373.687,A -85,B 0,C 180,E1 8317.728,E2 8317.728} C_VEL
LIN {X 0,Y 445.015,Z 389.923,A -85,B 0,C 180,E1 8320.49,E2 8320.49} C_VEL
LIN {X 0,Y 444.08,Z 401.619,A -85,B 0,C 180,E1 8323.591,E2 8323.591} C_VEL
LIN {X 0,Y 443.296,Z 408.615,A -85,B 0,C 180,E1 8327.094,E2 8327.094} C_VEL
LIN {X 0,Y 443.036,Z 410.147,A -85,B 0,C 180,E1 8329.674,E2 8329.674} C_VEL
LIN {X 0,Y 443.154,Z 408.104,A -85,B 0,C 180,E1 8332.761,E2 8332.761} C_VEL
LIN {X 0,Y 443.735,Z 401.311,A -85,B 0,C 180,E1 8335.974,E2 8335.974} C_VEL
LIN {X 0,Y 444.596,Z 389.445,A -85,B 0,C 180,E1 8339.091,E2 8339.091} C_VEL
LIN {X 0,Y 445.9,Z 371.397,A -85,B 0,C 180,E1 8342.079,E2 8342.079} C_VEL
LIN {X 0,Y 447.369,Z 349.212,A -85,B 0,C 180,E1 8344.476,E2 8344.476} C_VEL
LIN {X 0,Y 448.195,Z 325.373,A -85,B 0,C 180,E1 8346.171,E2 8346.171} C_VEL
LIN {X 0,Y 441.306,Z 297.81,A -85,B 0,C 180,E1 8347.723,E2 8347.723} C_VEL
LIN {X 0,Y 441.208,Z 297.81,A -85,B 0,C 180,E1 8354.121,E2 8354.121} C_VEL
LIN {X 0,Y 441.417,Z 297.81,A -85,B 0,C 180,E1 8359.1,E2 8359.1} C_VEL
LIN {X 0,Y 447.394,Z 326.659,A -85,B 0,C 180,E1 8360.323,E2 8360.323} C_VEL
LIN {X 0,Y 446.632,Z 350.318,A -85,B 0,C 180,E1 8361.867,E2 8361.867} C_VEL
LIN {X 0,Y 445.49,Z 372.267,A -85,B 0,C 180,E1 8364.168,E2 8364.168} C_VEL
LIN {X 0,Y 444.503,Z 388.835,A -85,B 0,C 180,E1 8366.838,E2 8366.838} C_VEL
LIN {X 0,Y 443.664,Z 401.183,A -85,B 0,C 180,E1 8370.001,E2 8370.001} C_VEL
LIN {X 0,Y 443.33,Z 407.548,A -85,B 0,C 180,E1 8372.927,E2 8372.927} C_VEL
LIN {X 0,Y 443.078,Z 409.862,A -85,B 0,C 180,E1 8375.865,E2 8375.865} C_VEL
LIN {X 0,Y 443.331,Z 407.857,A -85,B 0,C 180,E1 8379.128,E2 8379.128} C_VEL
LIN {X 0,Y 443.917,Z 401.149,A -85,B 0,C 180,E1 8382.267,E2 8382.267} C_VEL
LIN {X 0,Y 444.875,Z 388.367,A -85,B 0,C 180,E1 8385.514,E2 8385.514} C_VEL
LIN {X 0,Y 446.039,Z 371.195,A -85,B 0,C 180,E1 8388.244,E2 8388.244} C_VEL
LIN {X 0,Y 447.445,Z 349.484,A -85,B 0,C 180,E1 8390.467,E2 8390.467} C_VEL
LIN {X 0,Y 448.093,Z 325.498,A -85,B 0,C 180,E1 8392.002,E2 8392.002} C_VEL
LIN {X 0,Y 441.383,Z 299.734,A -85,B 0,C 180,E1 8393.179,E2 8393.179} C_VEL
LIN {X 0,Y 441.13,Z 297.81,A -85,B 0,C 180,E1 8393.287,E2 8393.287} C_VEL
LIN {X 0,Y 440.846,Z 297.81,A -85,B 0,C 180,E1 8398.635,E2 8398.635} C_VEL
LIN {X 0,Y 440.82,Z 297.81,A -85,B 0,C 180,E1 8405.588,E2 8405.588} C_VEL
LIN {X 0,Y 440.691,Z 297.81,A -85,B 0,C 180,E1 8411.101,E2 8411.101} C_VEL
LIN {X 0,Y 440.664,Z 297.81,A -85,B 0,C 180,E1 8416.756,E2 8416.756} C_VEL
LIN {X 0,Y 440.786,Z 297.81,A -85,B 0,C 180,E1 8421.943,E2 8421.943} C_VEL
LIN {X 0,Y 440.72,Z 297.81,A -85,B 0,C 180,E1 8426.766,E2 8426.766} C_VEL
LIN {X 0,Y 440.907,Z 297.81,A -85,B 0,C 180,E1 8433.567,E2 8433.567} C_VEL
LIN {X 0,Y 441.224,Z 297.81,A -85,B 0,C 180,E1 8439.987,E2 8439.987} C_VEL
LIN {X 0,Y 441.238,Z 297.81,A -85,B 0,C 180,E1 8446.136,E2 8446.136} C_VEL
LIN {X 0,Y 441.573,Z 297.81,A -85,B 0,C 180,E1 8452.979,E2 8452.979} C_VEL
LIN {X 0,Y 441.875,Z 297.81,A -85,B 0,C 180,E1 8459.988,E2 8459.988} C_VEL
LIN {X 0,Y 441.634,Z 297.81,A -85,B 0,C 180,E1 8465.871,E2 8465.871} C_VEL
LIN {X 0,Y 441.435,Z 297.81,A -85,B 0,C 180,E1 8471.823,E2 8471.823} C_VEL
LIN {X 0,Y 441.228,Z 297.81,A -85,B 0,C 180,E1 8477.914,E2 8477.914} C_VEL
LIN {X 0,Y 441.088,Z 297.81,A -85,B 0,C 180,E1 8484.225,E2 8484.225} C_VEL
LIN {X 0,Y 440.771,Z 297.81,A -85,B 0,C 180,E1 8491.141,E2 8491.141} C_VEL
LIN {X 0,Y 440.753,Z 297.81,A -85,B 0,C 180,E1 8495.579,E2 8495.579} C_VEL
LIN {X 0,Y 440.675,Z 297.81,A -85,B 0,C 180,E1 8501.118,E2 8501.118} C_VEL
LIN {X 0,Y 440.734,Z 297.81,A -85,B 0,C 180,E1 8506.782,E2 8506.782} C_VEL
LIN {X 0,Y 440.832,Z 297.81,A -85,B 0,C 180,E1 8511.964,E2 8511.964} C_VEL
LIN {X 0,Y 440.83,Z 297.81,A -85,B 0,C 180,E1 8518.824,E2 8518.824} C_VEL
LIN {X 0,Y 441.073,Z 297.81,A -85,B 0,C 180,E1 8521.918,E2 8521.918} C_VEL
LIN {X 0,Y 452.719,Z 335.973,A -85,B 0,C 180,E1 8523.163,E2 8523.163} C_VEL
LIN {X 0,Y 451.898,Z 376.057,A -85,B 0,C 180,E1 8524.002,E2 8524.002} C_VEL
LIN {X 0,Y 450.608,Z 397.529,A -85,B 0,C 180,E1 8524.853,E2 8524.853} C_VEL
LIN {X 0,Y 445.754,Z 413.497,A -85,B 0,C 180,E1 8525.559,E2 8525.559} C_VEL
LIN {X 0,Y 440.785,Z 428.773,A -85,B 0,C 180,E1 8526.462,E2 8526.462} C_VEL
LIN {X 0,Y 438.409,Z 457.691,A -85,B 0,C 180,E1 8529.138,E2 8529.138} C_VEL
LIN {X 0,Y 436.407,Z 482.553,A -85,B 0,C 180,E1 8532.388,E2 8532.388} C_VEL
LIN {X 0,Y 435.124,Z 503.681,A -85,B 0,C 180,E1 8536.274,E2 8536.274} C_VEL
LIN {X 0,Y 434.675,Z 517.789,A -85,B 0,C 180,E1 8540.004,E2 8540.004} C_VEL
LIN {X 0,Y 434.766,Z 527.607,A -85,B 0,C 180,E1 8544.023,E2 8544.023} C_VEL
LIN {X 0,Y 434.951,Z 532.28,A -85,B 0,C 180,E1 8548.011,E2 8548.011} C_VEL
LIN {X 0,Y 434.935,Z 532.189,A -85,B 0,C 180,E1 8551.988,E2 8551.988} C_VEL
LIN {X 0,Y 434.79,Z 527.353,A -85,B 0,C 180,E1 8555.976,E2 8555.976} C_VEL
LIN {X 0,Y 434.704,Z 517.405,A -85,B 0,C 180,E1 8559.995,E2 8559.995} C_VEL
LIN {X 0,Y 435.194,Z 501.712,A -85,B 0,C 180,E1 8564.046,E2 8564.046} C_VEL
LIN {X 0,Y 436.496,Z 480.296,A -85,B 0,C 180,E1 8567.867,E2 8567.867} C_VEL
LIN {X 0,Y 438.613,Z 454.158,A -85,B 0,C 180,E1 8571.185,E2 8571.185} C_VEL
LIN {X 0,Y 441.099,Z 424.447,A -85,B 0,C 180,E1 8573.834,E2 8573.834} C_VEL
LIN {X 0,Y 443.567,Z 392.358,A -85,B 0,C 180,E1 8575.729,E2 8575.729} C_VEL
LIN {X 0,Y 445.161,Z 359.289,A -85,B 0,C 180,E1 8576.845,E2 8576.845} C_VEL
LIN {X 0,Y 444.779,Z 333.045,A -85,B 0,C 180,E1 8577.342,E2 8577.342} C_VEL
LIN {X 0,Y 433.049,Z 297.81,A -85,B 0,C 180,E1 8578.664,E2 8578.664} C_VEL
LIN {X 0,Y 432.827,Z 297.81,A -85,B 0,C 180,E1 8583.904,E2 8583.904} C_VEL
LIN {X 0,Y 432.641,Z 297.81,A -85,B 0,C 180,E1 8589.902,E2 8589.902} C_VEL
LIN {X 0,Y 432.764,Z 297.81,A -85,B 0,C 180,E1 8597.074,E2 8597.074} C_VEL
LIN {X 0,Y 432.785,Z 297.81,A -85,B 0,C 180,E1 8603.662,E2 8603.662} C_VEL
LIN {X 0,Y 432.791,Z 297.81,A -85,B 0,C 180,E1 8608.48,E2 8608.48} C_VEL
LIN {X 0,Y 433.039,Z 297.81,A -85,B 0,C 180,E1 8615.294,E2 8615.294} C_VEL
LIN {X 0,Y 433.252,Z 297.81,A -85,B 0,C 180,E1 8621.744,E2 8621.744} C_VEL
LIN {X 0,Y 433.309,Z 297.81,A -85,B 0,C 180,E1 8627.952,E2 8627.952} C_VEL
LIN {X 0,Y 433.735,Z 297.81,A -85,B 0,C 180,E1 8634.021,E2 8634.021} C_VEL
LIN {X 0,Y 433.893,Z 297.81,A -85,B 0,C 180,E1 8640.012,E2 8640.012} C_VEL
LIN {X 0,Y 433.69,Z 297.81,A -85,B 0,C 180,E1 8646.004,E2 8646.004} C_VEL
LIN {X 0,Y 433.416,Z 297.81,A -85,B 0,C 180,E1 8652.878,E2 8652.878} C_VEL
LIN {X 0,Y 433.282,Z 297.81,A -85,B 0,C 180,E1 8658.281,E2 8658.281} C_VEL
LIN {X 0,Y 433.026,Z 297.81,A -85,B 0,C 180,E1 8665.038,E2 8665.038} C_VEL
LIN {X 0,Y 433.113,Z 297.81,A -85,B 0,C 180,E1 8671.243,E2 8671.243} C_VEL
LIN {X 0,Y 441.363,Z 327.369,A -85,B 0,C 180,E1 8673.033,E2 8673.033} C_VEL
LIN {X 0,Y 441.058,Z 347.548,A -85,B 0,C 180,E1 8674.491,E2 8674.491} C_VEL
LIN {X 0,Y 439.332,Z 369.692,A -85,B 0,C 180,E1 8676.784,E2 8676.784} C_VEL
LIN {X 0,Y 437.639,Z 388.371,A -85,B 0,C 180,E1 8679.738,E2 8679.738} C_VEL
LIN {X 0,Y 436.444,Z 401.484,A -85,B 0,C 180,E1 8683.028,E2 8683.028} C_VEL
LIN {X 0,Y 435.588,Z 409.354,A -85,B 0,C 180,E1 8686.697,E2 8686.697} C_VEL
LIN {X 0,Y 435.242,Z 411.251,A -85,B 0,C 180,E1 8689.728,E2 8689.728} C_VEL
LIN {X 0,Y 435.346,Z 409.071,A -85,B 0,C 180,E1 8692.889,E2 8692.889} C_VEL
LIN {X 0,Y 436.044,Z 401.492,A -85,B 0,C 180,E1 8696.379,E2 8696.379} C_VEL
LIN {X 0,Y 437.049,Z 388.251,A -85,B 0,C 180,E1 8699.702,E2 8699.702} C_VEL
LIN {X 0,Y 438.482,Z 369.9,A -85,B 0,C 180,E1 8702.623,E2 8702.623} C_VEL
LIN {X 0,Y 440.017,Z 347.703,A -85,B 0,C 180,E1 8704.96,E2 8704.96} C_VEL
LIN {X 0,Y 440.686,Z 327.037,A -85,B 0,C 180,E1 8706.43,E2 8706.43} C_VEL
LIN {X 0,Y 433.664,Z 299.906,A -85,B 0,C 180,E1 8707.967,E2 8707.967} C_VEL
LIN {X 0,Y 433.339,Z 297.81,A -85,B 0,C 180,E1 8708.151,E2 8708.151} C_VEL
LIN {X 0,Y 433.317,Z 297.81,A -85,B 0,C 180,E1 8713.824,E2 8713.824} C_VEL
LIN {X 0,Y 433.516,Z 298.423,A -85,B 0,C 180,E1 8718.857,E2 8718.857} C_VEL
LIN {X 0,Y 439.141,Z 323.729,A -85,B 0,C 180,E1 8719.857,E2 8719.857} C_VEL
LIN {X 0,Y 439.098,Z 347.927,A -85,B 0,C 180,E1 8721.365,E2 8721.365} C_VEL
LIN {X 0,Y 437.988,Z 370.079,A -85,B 0,C 180,E1 8723.572,E2 8723.572} C_VEL
LIN {X 0,Y 436.907,Z 387.773,A -85,B 0,C 180,E1 8726.288,E2 8726.288} C_VEL
LIN {X 0,Y 435.97,Z 401.017,A -85,B 0,C 180,E1 8729.505,E2 8729.505} C_VEL
LIN {X 0,Y 435.512,Z 408.742,A -85,B 0,C 180,E1 8732.98,E2 8732.98} C_VEL
LIN {X 0,Y 435.25,Z 410.958,A -85,B 0,C 180,E1 8735.971,E2 8735.971} C_VEL
LIN {X 0,Y 435.546,Z 408.824,A -85,B 0,C 180,E1 8739.292,E2 8739.292} C_VEL
LIN {X 0,Y 436.169,Z 402.007,A -85,B 0,C 180,E1 8742.488,E2 8742.488} C_VEL
LIN {X 0,Y 437.262,Z 388.928,A -85,B 0,C 180,E1 8745.816,E2 8745.816} C_VEL
LIN {X 0,Y 438.56,Z 371.036,A -85,B 0,C 180,E1 8748.645,E2 8748.645} C_VEL
LIN {X 0,Y 440.025,Z 349.422,A -85,B 0,C 180,E1 8750.843,E2 8750.843} C_VEL
LIN {X 0,Y 440.178,Z 324.578,A -85,B 0,C 180,E1 8752.436,E2 8752.436} C_VEL
LIN {X 0,Y 433.188,Z 297.81,A -85,B 0,C 180,E1 8753.667,E2 8753.667} C_VEL
LIN {X 0,Y 432.846,Z 297.81,A -85,B 0,C 180,E1 8759.332,E2 8759.332} C_VEL
LIN {X 0,Y 432.852,Z 297.81,A -85,B 0,C 180,E1 8763.904,E2 8763.904} C_VEL
LIN {X 0,Y 432.759,Z 297.81,A -85,B 0,C 180,E1 8769.882,E2 8769.882} C_VEL
LIN {X 0,Y 432.741,Z 297.81,A -85,B 0,C 180,E1 8775.761,E2 8775.761} C_VEL
LIN {X 0,Y 432.773,Z 297.81,A -85,B 0,C 180,E1 8781.107,E2 8781.107} C_VEL
LIN {X 0,Y 432.822,Z 297.81,A -85,B 0,C 180,E1 8786.798,E2 8786.798} C_VEL
LIN {X 0,Y 432.983,Z 297.81,A -85,B 0,C 180,E1 8793.045,E2 8793.045} C_VEL
LIN {X 0,Y 433.34,Z 297.81,A -85,B 0,C 180,E1 8800.088,E2 8800.088} C_VEL
LIN {X 0,Y 433.328,Z 297.81,A -85,B 0,C 180,E1 8807.178,E2 8807.178} C_VEL
LIN {X 0,Y 433.752,Z 297.81,A -85,B 0,C 180,E1 8813.997,E2 8813.997} C_VEL
LIN {X 0,Y 433.973,Z 297.81,A -85,B 0,C 180,E1 8819.988,E2 8819.988} C_VEL
LIN {X 0,Y 433.729,Z 297.81,A -85,B 0,C 180,E1 8825.979,E2 8825.979} C_VEL
LIN {X 0,Y 433.45,Z 297.81,A -85,B 0,C 180,E1 8832.893,E2 8832.893} C_VEL
LIN {X 0,Y 433.28,Z 297.81,A -85,B 0,C 180,E1 8838.254,E2 8838.254} C_VEL
LIN {X 0,Y 433.071,Z 297.81,A -85,B 0,C 180,E1 8845.048,E2 8845.048} C_VEL
LIN {X 0,Y 432.844,Z 297.81,A -85,B 0,C 180,E1 8851.516,E2 8851.516} C_VEL
LIN {X 0,Y 432.734,Z 297.81,A -85,B 0,C 180,E1 8858.865,E2 8858.865} C_VEL
LIN {X 0,Y 432.799,Z 297.81,A -85,B 0,C 180,E1 8865.787,E2 8865.787} C_VEL
LIN {X 0,Y 432.85,Z 297.81,A -85,B 0,C 180,E1 8871.132,E2 8871.132} C_VEL
LIN {X 0,Y 432.902,Z 297.81,A -85,B 0,C 180,E1 8878.475,E2 8878.475} C_VEL
LIN {X 0,Y 433.168,Z 298.334,A -85,B 0,C 180,E1 8881.528,E2 8881.528} C_VEL
LIN {X 0,Y 445.295,Z 335.474,A -85,B 0,C 180,E1 8882.783,E2 8882.783} C_VEL
LIN {X 0,Y 444.511,Z 375.678,A -85,B 0,C 180,E1 8883.642,E2 8883.642} C_VEL
LIN {X 0,Y 442.422,Z 407.663,A -85,B 0,C 180,E1 8885.064,E2 8885.064} C_VEL
LIN {X 0,Y 440.785,Z 428.773,A -85,B 0,C 180,E1 8886.462,E2 8886.462} C_VEL
LIN {X 0,Y 435.634,Z 443.504,A -85,B 0,C 180,E1 8887.571,E2 8887.571} C_VEL
LIN {X 0,Y 430.715,Z 457.04,A -85,B 0,C 180,E1 8888.853,E2 8888.853} C_VEL
LIN {X 0,Y 428.569,Z 482.407,A -85,B 0,C 180,E1 8892.251,E2 8892.251} C_VEL
LIN {X 0,Y 427.293,Z 502.442,A -85,B 0,C 180,E1 8896.017,E2 8896.017} C_VEL
LIN {X 0,Y 426.805,Z 518.178,A -85,B 0,C 180,E1 8900.332,E2 8900.332} C_VEL
LIN {X 0,Y 426.913,Z 526.488,A -85,B 0,C 180,E1 8903.912,E2 8903.912} C_VEL
LIN {X 0,Y 427.123,Z 531.183,A -85,B 0,C 180,E1 8907.975,E2 8907.975} C_VEL
LIN {X 0,Y 427.107,Z 531.093,A -85,B 0,C 180,E1 8912.024,E2 8912.024} C_VEL
LIN {X 0,Y 426.943,Z 526.24,A -85,B 0,C 180,E1 8916.086,E2 8916.086} C_VEL
LIN {X 0,Y 426.849,Z 516.256,A -85,B 0,C 180,E1 8920.181,E2 8920.181} C_VEL
LIN {X 0,Y 427.351,Z 500.519,A -85,B 0,C 180,E1 8924.31,E2 8924.31} C_VEL
LIN {X 0,Y 428.796,Z 479.051,A -85,B 0,C 180,E1 8928.198,E2 8928.198} C_VEL
LIN {X 0,Y 431.078,Z 452.699,A -85,B 0,C 180,E1 8931.586,E2 8931.586} C_VEL
LIN {X 0,Y 433.7,Z 422.901,A -85,B 0,C 180,E1 8934.267,E2 8934.267} C_VEL
LIN {X 0,Y 436.282,Z 391.266,A -85,B 0,C 180,E1 8936.149,E2 8936.149} C_VEL
LIN {X 0,Y 437.938,Z 358.135,A -85,B 0,C 180,E1 8937.275,E2 8937.275} C_VEL
LIN {X 0,Y 437.584,Z 334.718,A -85,B 0,C 180,E1 8937.729,E2 8937.729} C_VEL
LIN {X 0,Y 425.083,Z 297.81,A -85,B 0,C 180,E1 8939.241,E2 8939.241} C_VEL
LIN {X 0,Y 424.807,Z 297.81,A -85,B 0,C 180,E1 8945.233,E2 8945.233} C_VEL
LIN {X 0,Y 424.749,Z 297.81,A -85,B 0,C 180,E1 8951.767,E2 8951.767} C_VEL
LIN {X 0,Y 424.849,Z 297.81,A -85,B 0,C 180,E1 8958.234,E2 8958.234} C_VEL
LIN {X 0,Y 424.828,Z 297.81,A -85,B 0,C 180,E1 8964.781,E2 8964.781} C_VEL
LIN {X 0,Y 424.914,Z 297.81,A -85,B 0,C 180,E1 8970.2,E2 8970.2} C_VEL
LIN {X 0,Y 425.234,Z 297.81,A -85,B 0,C 180,E1 8977.314,E2 8977.314} C_VEL
LIN {X 0,Y 425.309,Z 297.81,A -85,B 0,C 180,E1 8983.523,E2 8983.523} C_VEL
LIN {X 0,Y 425.488,Z 297.81,A -85,B 0,C 180,E1 8989.799,E2 8989.799} C_VEL
LIN {X 0,Y 425.849,Z 297.81,A -85,B 0,C 180,E1 8995.949,E2 8995.949} C_VEL
LIN {X 0,Y 425.888,Z 297.81,A -85,B 0,C 180,E1 9002.043,E2 9002.043} C_VEL
LIN {X 0,Y 425.695,Z 297.81,A -85,B 0,C 180,E1 9008.165,E2 9008.165} C_VEL
LIN {X 0,Y 425.498,Z 297.81,A -85,B 0,C 180,E1 9014.388,E2 9014.388} C_VEL
LIN {X 0,Y 425.277,Z 297.81,A -85,B 0,C 180,E1 9020.797,E2 9020.797} C_VEL
LIN {X 0,Y 425.083,Z 297.81,A -85,B 0,C 180,E1 9027.498,E2 9027.498} C_VEL
LIN {X 0,Y 425.188,Z 297.81,A -85,B 0,C 180,E1 9030.765,E2 9030.765} C_VEL
LIN {X 0,Y 433.15,Z 325.284,A -85,B 0,C 180,E1 9032.428,E2 9032.428} C_VEL
LIN {X 0,Y 434.47,Z 338.024,A -85,B 0,C 180,E1 9033.344,E2 9033.344} C_VEL
LIN {X 0,Y 432.689,Z 361.352,A -85,B 0,C 180,E1 9035.384,E2 9035.384} C_VEL
LIN {X 0,Y 430.786,Z 381.27,A -85,B 0,C 180,E1 9038.027,E2 9038.027} C_VEL
LIN {X 0,Y 429.164,Z 397.174,A -85,B 0,C 180,E1 9041.262,E2 9041.262} C_VEL
LIN {X 0,Y 428.157,Z 407.543,A -85,B 0,C 180,E1 9044.839,E2 9044.839} C_VEL
LIN {X 0,Y 427.558,Z 411.712,A -85,B 0,C 180,E1 9047.889,E2 9047.889} C_VEL
LIN {X 0,Y 427.391,Z 411.998,A -85,B 0,C 180,E1 9050.987,E2 9050.987} C_VEL
LIN {X 0,Y 427.751,Z 407.995,A -85,B 0,C 180,E1 9054.255,E2 9054.255} C_VEL
LIN {X 0,Y 428.577,Z 398.549,A -85,B 0,C 180,E1 9057.701,E2 9057.701} C_VEL
LIN {X 0,Y 429.824,Z 383.204,A -85,B 0,C 180,E1 9061.009,E2 9061.009} C_VEL
LIN {X 0,Y 431.431,Z 363.093,A -85,B 0,C 180,E1 9063.812,E2 9063.812} C_VEL
LIN {X 0,Y 432.998,Z 339.511,A -85,B 0,C 180,E1 9065.965,E2 9065.965} C_VEL
LIN {X 0,Y 432.575,Z 325.953,A -85,B 0,C 180,E1 9066.894,E2 9066.894} C_VEL
LIN {X 0,Y 425.438,Z 297.81,A -85,B 0,C 180,E1 9068.545,E2 9068.545} C_VEL
LIN {X 0,Y 425.335,Z 297.81,A -85,B 0,C 180,E1 9075.621,E2 9075.621} C_VEL
LIN {X 0,Y 425.559,Z 297.81,A -85,B 0,C 180,E1 9078.53,E2 9078.53} C_VEL
LIN {X 0,Y 431.64,Z 325.552,A -85,B 0,C 180,E1 9079.642,E2 9079.642} C_VEL
LIN {X 0,Y 431.472,Z 349.779,A -85,B 0,C 180,E1 9081.199,E2 9081.199} C_VEL
LIN {X 0,Y 430.271,Z 371.743,A -85,B 0,C 180,E1 9083.456,E2 9083.456} C_VEL
LIN {X 0,Y 429.142,Z 389.225,A -85,B 0,C 180,E1 9086.22,E2 9086.22} C_VEL
LIN {X 0,Y 428.154,Z 402.317,A -85,B 0,C 180,E1 9089.496,E2 9089.496} C_VEL
LIN {X 0,Y 427.672,Z 409.935,A -85,B 0,C 180,E1 9093.034,E2 9093.034} C_VEL
LIN {X 0,Y 427.424,Z 412.053,A -85,B 0,C 180,E1 9096.08,E2 9096.08} C_VEL
LIN {X 0,Y 427.667,Z 410.604,A -85,B 0,C 180,E1 9098.805,E2 9098.805} C_VEL
LIN {X 0,Y 428.368,Z 404.312,A -85,B 0,C 180,E1 9102.203,E2 9102.203} C_VEL
LIN {X 0,Y 429.409,Z 392.037,A -85,B 0,C 180,E1 9105.61,E2 9105.61} C_VEL
LIN {X 0,Y 430.81,Z 374.642,A -85,B 0,C 180,E1 9108.571,E2 9108.571} C_VEL
LIN {X 0,Y 432.367,Z 353.42,A -85,B 0,C 180,E1 9110.89,E2 9110.89} C_VEL
LIN {X 0,Y 433.174,Z 328.362,A -85,B 0,C 180,E1 9112.6,E2 9112.6} C_VEL
LIN {X 0,Y 426.634,Z 303.286,A -85,B 0,C 180,E1 9113.833,E2 9113.833} C_VEL
LIN {X 0,Y 425.286,Z 297.81,A -85,B 0,C 180,E1 9114.037,E2 9114.037} C_VEL
LIN {X 0,Y 424.896,Z 297.81,A -85,B 0,C 180,E1 9119.816,E2 9119.816} C_VEL
LIN {X 0,Y 424.862,Z 297.81,A -85,B 0,C 180,E1 9127.143,E2 9127.143} C_VEL
LIN {X 0,Y 424.819,Z 297.81,A -85,B 0,C 180,E1 9132.447,E2 9132.447} C_VEL
LIN {X 0,Y 424.859,Z 297.81,A -85,B 0,C 180,E1 9138.235,E2 9138.235} C_VEL
LIN {X 0,Y 424.834,Z 297.81,A -85,B 0,C 180,E1 9145.351,E2 9145.351} C_VEL
LIN {X 0,Y 424.885,Z 297.81,A -85,B 0,C 180,E1 9150.168,E2 9150.168} C_VEL
LIN {X 0,Y 425.239,Z 297.81,A -85,B 0,C 180,E1 9157.315,E2 9157.315} C_VEL
LIN {X 0,Y 425.369,Z 297.81,A -85,B 0,C 180,E1 9163.499,E2 9163.499} C_VEL
LIN {X 0,Y 425.543,Z 297.81,A -85,B 0,C 180,E1 9169.774,E2 9169.774} C_VEL
LIN {X 0,Y 425.858,Z 297.81,A -85,B 0,C 180,E1 9175.923,E2 9175.923} C_VEL
LIN {X 0,Y 425.931,Z 297.81,A -85,B 0,C 180,E1 9182.018,E2 9182.018} C_VEL
LIN {X 0,Y 425.7,Z 297.81,A -85,B 0,C 180,E1 9188.139,E2 9188.139} C_VEL
LIN {X 0,Y 425.514,Z 297.81,A -85,B 0,C 180,E1 9194.361,E2 9194.361} C_VEL
LIN {X 0,Y 425.292,Z 297.81,A -85,B 0,C 180,E1 9200.769,E2 9200.769} C_VEL
LIN {X 0,Y 425.074,Z 297.81,A -85,B 0,C 180,E1 9207.47,E2 9207.47} C_VEL
LIN {X 0,Y 424.919,Z 297.81,A -85,B 0,C 180,E1 9212.173,E2 9212.173} C_VEL
LIN {X 0,Y 424.805,Z 297.81,A -85,B 0,C 180,E1 9218.602,E2 9218.602} C_VEL
LIN {X 0,Y 424.872,Z 297.81,A -85,B 0,C 180,E1 9225.246,E2 9225.246} C_VEL
LIN {X 0,Y 424.921,Z 297.81,A -85,B 0,C 180,E1 9231.359,E2 9231.359} C_VEL
LIN {X 0,Y 424.997,Z 297.81,A -85,B 0,C 180,E1 9238.424,E2 9238.424} C_VEL
LIN {X 0,Y 425.158,Z 297.81,A -85,B 0,C 180,E1 9241.062,E2 9241.062} C_VEL
LIN {X 0,Y 437.984,Z 337.722,A -85,B 0,C 180,E1 9242.441,E2 9242.441} C_VEL
LIN {X 0,Y 437.108,Z 375.861,A -85,B 0,C 180,E1 9243.29,E2 9243.29} C_VEL
LIN {X 0,Y 434.881,Z 408.322,A -85,B 0,C 180,E1 9244.784,E2 9244.784} C_VEL
LIN {X 0,Y 432.386,Z 438.708,A -85,B 0,C 180,E1 9247.018,E2 9247.018} C_VEL
LIN {X 0,Y 430.715,Z 457.04,A -85,B 0,C 180,E1 9248.853,E2 9248.853} C_VEL
LIN {X 0,Y 425.727,Z 469.767,A -85,B 0,C 180,E1 9250.327,E2 9250.327} C_VEL
LIN {X 0,Y 420.814,Z 481.386,A -85,B 0,C 180,E1 9251.972,E2 9251.972} C_VEL
LIN {X 0,Y 419.418,Z 501.938,A -85,B 0,C 180,E1 9255.925,E2 9255.925} C_VEL
LIN {X 0,Y 418.933,Z 517.009,A -85,B 0,C 180,E1 9260.148,E2 9260.148} C_VEL
LIN {X 0,Y 419.057,Z 525.363,A -85,B 0,C 180,E1 9263.798,E2 9263.798} C_VEL
LIN {X 0,Y 419.302,Z 530.085,A -85,B 0,C 180,E1 9267.937,E2 9267.937} C_VEL
LIN {X 0,Y 419.288,Z 529.997,A -85,B 0,C 180,E1 9272.062,E2 9272.062} C_VEL
LIN {X 0,Y 419.09,Z 525.128,A -85,B 0,C 180,E1 9276.201,E2 9276.201} C_VEL
LIN {X 0,Y 418.983,Z 515.112,A -85,B 0,C 180,E1 9280.374,E2 9280.374} C_VEL
LIN {X 0,Y 419.526,Z 499.34,A -85,B 0,C 180,E1 9284.582,E2 9284.582} C_VEL
LIN {X 0,Y 421.054,Z 477.807,A -85,B 0,C 180,E1 9288.545,E2 9288.545} C_VEL
LIN {X 0,Y 423.43,Z 452.317,A -85,B 0,C 180,E1 9291.886,E2 9291.886} C_VEL
LIN {X 0,Y 426.167,Z 423.151,A -85,B 0,C 180,E1 9294.585,E2 9294.585} C_VEL
LIN {X 0,Y 428.956,Z 391.221,A -85,B 0,C 180,E1 9296.538,E2 9296.538} C_VEL
LIN {X 0,Y 430.732,Z 357.942,A -85,B 0,C 180,E1 9297.699,E2 9297.699} C_VEL
LIN {X 0,Y 430.226,Z 335.921,A -85,B 0,C 180,E1 9298.154,E2 9298.154} C_VEL
LIN {X 0,Y 417.12,Z 297.81,A -85,B 0,C 180,E1 9299.768,E2 9299.768} C_VEL
LIN {X 0,Y 416.918,Z 297.81,A -85,B 0,C 180,E1 9307.244,E2 9307.244} C_VEL
LIN {X 0,Y 416.781,Z 297.81,A -85,B 0,C 180,E1 9313.621,E2 9313.621} C_VEL
LIN {X 0,Y 416.882,Z 297.81,A -85,B 0,C 180,E1 9319.476,E2 9319.476} C_VEL
LIN {X 0,Y 416.914,Z 297.81,A -85,B 0,C 180,E1 9324.627,E2 9324.627} C_VEL
LIN {X 0,Y 417.038,Z 297.81,A -85,B 0,C 180,E1 9331.954,E2 9331.954} C_VEL
LIN {X 0,Y 417.329,Z 297.81,A -85,B 0,C 180,E1 9338.816,E2 9338.816} C_VEL
LIN {X 0,Y 417.387,Z 297.81,A -85,B 0,C 180,E1 9345.353,E2 9345.353} C_VEL
LIN {X 0,Y 417.721,Z 297.81,A -85,B 0,C 180,E1 9351.705,E2 9351.705} C_VEL
LIN {X 0,Y 418.181,Z 297.81,A -85,B 0,C 180,E1 9357.945,E2 9357.945} C_VEL
LIN {X 0,Y 417.957,Z 297.81,A -85,B 0,C 180,E1 9364.154,E2 9364.154} C_VEL
LIN {X 0,Y 417.685,Z 297.81,A -85,B 0,C 180,E1 9370.42,E2 9370.42} C_VEL
LIN {X 0,Y 417.5,Z 297.81,A -85,B 0,C 180,E1 9376.821,E2 9376.821} C_VEL
LIN {X 0,Y 417.238,Z 297.81,A -85,B 0,C 180,E1 9383.457,E2 9383.457} C_VEL
LIN {X 0,Y 417.293,Z 298.598,A -85,B 0,C 180,E1 9390.275,E2 9390.275} C_VEL
LIN {X 0,Y 425.638,Z 326.3,A -85,B 0,C 180,E1 9392.022,E2 9392.022} C_VEL
LIN {X 0,Y 427.226,Z 337.96,A -85,B 0,C 180,E1 9392.897,E2 9392.897} C_VEL
LIN {X 0,Y 425.359,Z 361.075,A -85,B 0,C 180,E1 9394.915,E2 9394.915} C_VEL
LIN {X 0,Y 423.379,Z 381.022,A -85,B 0,C 180,E1 9397.541,E2 9397.541} C_VEL
LIN {X 0,Y 421.579,Z 397.359,A -85,B 0,C 180,E1 9400.817,E2 9400.817} C_VEL
LIN {X 0,Y 420.558,Z 407.454,A -85,B 0,C 180,E1 9404.143,E2 9404.143} C_VEL
LIN {X 0,Y 419.903,Z 412.035,A -85,B 0,C 180,E1 9406.938,E2 9406.938} C_VEL
LIN {X 0,Y 419.587,Z 413.461,A -85,B 0,C 180,E1 9409.659,E2 9409.659} C_VEL
LIN {X 0,Y 419.796,Z 410.534,A -85,B 0,C 180,E1 9413.47,E2 9413.47} C_VEL
LIN {X 0,Y 420.599,Z 402.332,A -85,B 0,C 180,E1 9417.012,E2 9417.012} C_VEL
LIN {X 0,Y 421.779,Z 388.592,A -85,B 0,C 180,E1 9420.401,E2 9420.401} C_VEL
LIN {X 0,Y 423.476,Z 368.815,A -85,B 0,C 180,E1 9423.496,E2 9423.496} C_VEL
LIN {X 0,Y 425.263,Z 344.573,A -85,B 0,C 180,E1 9425.947,E2 9425.947} C_VEL
LIN {X 0,Y 425.474,Z 329.418,A -85,B 0,C 180,E1 9427.038,E2 9427.038} C_VEL
LIN {X 0,Y 418.632,Z 302.603,A -85,B 0,C 180,E1 9428.665,E2 9428.665} C_VEL
LIN {X 0,Y 417.509,Z 297.81,A -85,B 0,C 180,E1 9428.986,E2 9428.986} C_VEL
LIN {X 0,Y 417.409,Z 297.81,A -85,B 0,C 180,E1 9435.342,E2 9435.342} C_VEL
LIN {X 0,Y 417.624,Z 297.81,A -85,B 0,C 180,E1 9438.21,E2 9438.21} C_VEL
LIN {X 0,Y 423.716,Z 325.161,A -85,B 0,C 180,E1 9439.296,E2 9439.296} C_VEL
LIN {X 0,Y 424.185,Z 343.475,A -85,B 0,C 180,E1 9440.401,E2 9440.401} C_VEL
LIN {X 0,Y 422.969,Z 366.107,A -85,B 0,C 180,E1 9442.441,E2 9442.441} C_VEL
LIN {X 0,Y 421.781,Z 385.232,A -85,B 0,C 180,E1 9445.126,E2 9445.126} C_VEL
LIN {X 0,Y 420.672,Z 400.321,A -85,B 0,C 180,E1 9448.459,E2 9448.459} C_VEL
LIN {X 0,Y 419.946,Z 409.55,A -85,B 0,C 180,E1 9452.06,E2 9452.06} C_VEL
LIN {X 0,Y 419.707,Z 412.204,A -85,B 0,C 180,E1 9454.124,E2 9454.124} C_VEL
LIN {X 0,Y 419.599,Z 413.141,A -85,B 0,C 180,E1 9456.194,E2 9456.194} C_VEL
